C05422=1058.891,318.476,-103.732,173.436,35.812,156.715
C05423=1058.885,318.224,-103.698,173.433,35.808,156.714
C05424=1058.878,317.971,-103.663,173.428,35.803,156.713
C05425=1058.871,317.718,-103.629,173.425,35.799,156.712
C05426=1058.864,317.467,-103.595,173.421,35.795,156.711
C05427=1058.859,317.219,-103.561,173.418,35.790,156.711
C05428=1058.852,316.971,-103.527,173.414,35.786,156.710
C05429=1058.846,316.723,-103.494,173.411,35.782,156.709
C05430=1058.839,316.476,-103.460,173.408,35.778,156.708
C05431=1058.833,316.228,-103.426,173.404,35.773,156.707
C05432=1058.827,315.981,-103.393,173.401,35.769,156.706
C05433=1058.820,315.733,-103.359,173.397,35.765,156.705
C05434=1058.814,315.485,-103.326,173.394,35.760,156.704
C05435=1058.808,315.238,-103.292,173.391,35.756,156.703
C05436=1058.801,314.989,-103.259,173.388,35.752,156.702
C05437=1058.795,314.742,-103.225,173.384,35.748,156.701
C05438=1058.789,314.495,-103.192,173.381,35.744,156.700
C05439=1058.783,314.247,-103.158,173.378,35.740,156.699
C05440=1058.776,313.999,-103.125,173.374,35.735,156.698
C05441=1058.770,313.752,-103.091,173.371,35.731,156.698
C05442=1058.763,313.503,-103.058,173.367,35.727,156.697
C05443=1058.757,313.256,-103.025,173.364,35.723,156.696
C05444=1058.751,313.009,-102.992,173.360,35.719,156.695
C05445=1058.744,312.761,-102.959,173.357,35.715,156.694
C05446=1058.737,312.513,-102.926,173.354,35.711,156.693
C05447=1058.730,312.265,-102.892,173.350,35.706,156.692
C05448=1058.724,312.018,-102.859,173.347,35.702,156.691
C05449=1058.717,311.770,-102.827,173.343,35.698,156.691
C05450=1058.710,311.522,-102.794,173.340,35.694,156.690
C05451=1058.704,311.275,-102.761,173.337,35.690,156.689
C05452=1058.697,311.028,-102.728,173.333,35.686,156.688
C05453=1058.690,310.779,-102.695,173.330,35.682,156.687
C05454=1058.684,310.532,-102.662,173.326,35.678,156.686
C05455=1058.678,310.284,-102.629,173.323,35.674,156.685
C05456=1058.671,310.036,-102.596,173.320,35.670,156.684
C05457=1058.664,309.788,-102.563,173.316,35.666,156.684
C05458=1058.658,309.541,-102.531,173.314,35.662,156.683
C05459=1058.652,309.293,-102.498,173.310,35.658,156.682
C05460=1058.645,309.045,-102.465,173.307,35.654,156.681
C05461=1058.639,308.797,-102.432,173.303,35.650,156.680
C05462=1058.631,308.551,-102.399,173.300,35.645,156.679
C05463=1058.625,308.302,-102.367,173.297,35.642,156.679
C05464=1058.618,308.054,-102.334,173.293,35.638,156.678
C05465=1058.612,307.806,-102.301,173.290,35.634,156.677
C05466=1058.606,307.559,-102.269,173.287,35.630,156.676
C05467=1058.600,307.311,-102.236,173.283,35.626,156.675
C05468=1058.593,307.064,-102.203,173.280,35.622,156.674
C05469=1058.586,306.815,-102.170,173.277,35.617,156.673
C05470=1058.579,306.568,-102.138,173.274,35.613,156.672
C05471=1058.573,306.320,-102.105,173.271,35.609,156.672
C05472=1058.567,306.073,-102.072,173.267,35.605,156.671
C05473=1058.560,305.825,-102.040,173.264,35.601,156.670
C05474=1058.554,305.578,-102.007,173.260,35.598,156.669
C05475=1058.548,305.329,-101.975,173.257,35.594,156.668
C05476=1058.541,305.081,-101.942,173.255,35.590,156.667
C05477=1058.534,304.834,-101.910,173.251,35.585,156.666
C05478=1058.528,304.586,-101.877,173.248,35.581,156.666
C05479=1058.522,304.338,-101.845,173.244,35.577,156.665
C05480=1058.515,304.090,-101.812,173.241,35.573,156.664
C05481=1058.509,303.842,-101.780,173.238,35.569,156.663
C05482=1058.503,303.593,-101.746,173.234,35.566,156.662
C05483=1058.496,303.345,-101.715,173.232,35.561,156.661
C05484=1058.490,303.097,-101.682,173.228,35.557,156.660
C05485=1058.484,302.850,-101.649,173.225,35.553,156.660
C05486=1058.478,302.602,-101.617,173.222,35.549,156.659
C05487=1058.471,302.354,-101.584,173.218,35.545,156.658
C05488=1058.464,302.107,-101.552,173.216,35.541,156.657
C05489=1058.458,301.859,-101.520,173.213,35.538,156.656
C05490=1058.452,301.611,-101.487,173.209,35.533,156.655
C05491=1058.446,301.363,-101.455,173.206,35.529,156.655
C05492=1058.440,301.115,-101.423,173.202,35.525,156.654
C05493=1058.433,300.867,-101.391,173.200,35.521,156.653
C05494=1058.427,300.620,-101.358,173.197,35.517,156.652
C05495=1058.420,300.372,-101.326,173.193,35.514,156.651
C05496=1058.414,300.124,-101.294,173.190,35.509,156.650
C05497=1058.408,299.876,-101.261,173.187,35.505,156.649
C05498=1058.401,299.628,-101.230,173.184,35.501,156.649
C05499=1058.395,299.380,-101.198,173.181,35.497,156.648
C05500=1058.389,299.133,-101.165,173.177,35.494,156.647
C05501=1058.383,298.884,-101.133,173.174,35.490,156.646
C05502=1058.377,298.638,-101.101,173.172,35.485,156.645
C05503=1058.371,298.390,-101.069,173.168,35.481,156.644
C05504=1058.364,298.142,-101.036,173.165,35.477,156.644
C05505=1058.358,297.894,-101.004,173.162,35.474,156.643
C05506=1058.352,297.646,-100.973,173.159,35.470,156.642
C05507=1058.345,297.398,-100.940,173.156,35.466,156.641
C05508=1058.339,297.150,-100.908,173.152,35.461,156.640
C05509=1058.334,296.903,-100.876,173.150,35.457,156.639
C05510=1058.327,296.655,-100.844,173.147,35.454,156.639
C05511=1058.321,296.407,-100.812,173.143,35.450,156.638
C05512=1058.314,296.159,-100.781,173.140,35.446,156.637
C05513=1058.308,295.911,-100.749,173.138,35.442,156.636
C05514=1058.302,295.663,-100.717,173.134,35.438,156.635
C05515=1058.295,295.415,-100.685,173.131,35.434,156.635
C05516=1058.289,295.168,-100.653,173.128,35.430,156.634
C05517=1058.283,294.919,-100.621,173.125,35.426,156.633
C05518=1058.276,294.672,-100.590,173.122,35.423,156.632
C05519=1058.270,294.424,-100.559,173.119,35.419,156.631
C05520=1058.264,294.176,-100.527,173.115,35.415,156.630
C05521=1058.257,293.928,-100.495,173.113,35.411,156.630
C05522=1058.250,293.680,-100.464,173.110,35.407,156.629
C05523=1058.244,293.432,-100.432,173.106,35.403,156.628
C05524=1058.238,293.185,-100.401,173.104,35.399,156.627
C05525=1058.232,292.937,-100.369,173.101,35.396,156.626
C05526=1058.226,292.689,-100.337,173.097,35.392,156.626
C05527=1058.219,292.441,-100.306,173.095,35.388,156.625
C05528=1058.213,292.193,-100.274,173.092,35.384,156.624
C05529=1058.206,291.945,-100.242,173.088,35.380,156.623
C05530=1058.200,291.697,-100.211,173.086,35.376,156.622
C05531=1058.194,291.457,-100.180,173.083,35.373,156.622
C05532=1058.188,291.217,-100.150,173.079,35.369,156.621
C05533=1058.182,290.976,-100.119,173.077,35.365,156.620
C05534=1058.175,290.736,-100.089,173.074,35.362,156.619
C05535=1058.169,290.496,-100.058,173.071,35.358,156.619
C05536=1058.163,290.255,-100.028,173.068,35.354,156.618
C05537=1058.156,290.015,-99.998,173.065,35.350,156.617
C05538=1058.151,289.774,-99.967,173.062,35.347,156.616
C05539=1058.144,289.527,-99.936,173.059,35.343,156.615
C05540=1058.138,289.279,-99.905,173.057,35.339,156.615
C05541=1058.132,289.031,-99.872,173.053,35.335,156.614
C05542=1058.126,288.783,-99.842,173.050,35.332,156.613
C05543=1058.119,288.535,-99.811,173.048,35.327,156.612
C05544=1058.112,288.287,-99.779,173.044,35.324,156.611
C05545=1058.106,288.039,-99.749,173.041,35.320,156.611
C05546=1058.100,287.791,-99.717,173.039,35.316,156.610
C05547=1058.094,287.543,-99.685,173.035,35.313,156.609
C05548=1058.088,287.295,-99.655,173.032,35.309,156.608
C05549=1058.081,287.047,-99.623,173.030,35.305,156.607
C05550=1058.075,286.800,-99.592,173.026,35.301,156.607
C05551=1058.068,286.551,-99.562,173.024,35.297,156.606
C05552=1058.062,286.303,-99.530,173.021,35.294,156.605
C05553=1058.056,286.055,-99.500,173.017,35.290,156.604
C05554=1058.049,285.807,-99.468,173.015,35.286,156.604
C05555=1058.042,285.560,-99.437,173.012,35.282,156.603
C05556=1058.036,285.312,-99.407,173.008,35.278,156.602
C05557=1058.030,285.064,-99.375,173.006,35.275,156.601
C05558=1058.023,284.815,-99.344,173.003,35.271,156.600
C05559=1058.017,284.568,-99.313,173.001,35.267,156.600
C05560=1058.011,284.320,-99.283,172.997,35.263,156.599
C05561=1058.004,284.071,-99.252,172.994,35.260,156.598
C05562=1057.998,283.824,-99.221,172.992,35.256,156.597
C05563=1057.992,283.575,-99.190,172.988,35.252,156.596
C05564=1057.986,283.328,-99.159,172.986,35.248,156.596
C05565=1057.979,283.080,-99.128,172.983,35.245,156.595
C05566=1057.973,282.832,-99.097,172.980,35.241,156.594
C05567=1057.967,282.584,-99.067,172.977,35.237,156.593
C05568=1057.960,282.335,-99.036,172.974,35.233,156.593
C05569=1057.954,282.088,-99.005,172.971,35.229,156.592
C05570=1057.948,281.840,-98.974,172.968,35.226,156.591
C05571=1057.942,281.592,-98.944,172.966,35.222,156.590
C05572=1057.935,281.344,-98.912,172.962,35.218,156.590
C05573=1057.929,281.096,-98.882,172.960,35.215,156.589
C05574=1057.923,280.848,-98.851,172.957,35.210,156.588
C05575=1057.917,280.600,-98.821,172.955,35.207,156.587
C05576=1057.910,280.352,-98.789,172.951,35.203,156.586
C05577=1057.905,280.104,-98.759,172.949,35.199,156.586
C05578=1057.898,279.856,-98.728,172.946,35.196,156.585
C05579=1057.892,279.608,-98.698,172.942,35.192,156.584
C05580=1057.885,279.359,-98.668,172.940,35.188,156.583
C05581=1057.879,279.112,-98.636,172.937,35.184,156.583
C05582=1057.873,278.864,-98.606,172.934,35.181,156.582
C05583=1057.866,278.615,-98.575,172.931,35.177,156.581
C05584=1057.860,278.368,-98.546,172.929,35.173,156.580
C05585=1057.853,278.119,-98.515,172.926,35.170,156.580
C05586=1057.847,277.871,-98.485,172.923,35.165,156.579
C05587=1057.842,277.637,-98.456,172.920,35.162,156.578
C05588=1057.836,277.401,-98.427,172.918,35.159,156.577
C05589=1057.830,277.166,-98.398,172.915,35.155,156.577
C05590=1057.824,276.932,-98.369,172.912,35.152,156.576
C05591=1057.817,276.697,-98.341,172.910,35.148,156.575
C05592=1057.811,276.462,-98.312,172.907,35.145,156.574
C05593=1057.806,276.227,-98.283,172.904,35.141,156.574
C05594=1057.800,275.992,-98.255,172.902,35.138,156.573
C05595=1057.794,275.744,-98.224,172.899,35.134,156.572
C05596=1057.787,275.496,-98.194,172.896,35.130,156.571
C05597=1057.781,275.248,-98.163,172.893,35.126,156.571
C05598=1057.775,275.000,-98.133,172.891,35.123,156.570
C05599=1057.764,274.601,-98.084,172.886,35.117,156.569
C05600=1057.754,274.203,-98.036,172.882,35.111,156.568
C05601=1057.744,273.805,-97.988,172.877,35.105,156.566
C05602=1057.734,273.406,-97.940,172.873,35.099,156.565
C05603=1057.728,273.158,-97.909,172.870,35.095,156.564
C05604=1057.722,272.911,-97.879,172.867,35.091,156.564
C05605=1057.715,272.662,-97.849,172.865,35.088,156.563
C05606=1057.710,272.414,-97.819,172.862,35.084,156.562
C05607=1057.703,272.166,-97.789,172.860,35.081,156.561
C05608=1057.697,271.918,-97.759,172.856,35.076,156.560
C05609=1057.690,271.670,-97.730,172.854,35.073,156.560
C05610=1057.684,271.421,-97.699,172.851,35.069,156.559
C05611=1057.678,271.173,-97.669,172.849,35.066,156.558
C05612=1057.672,270.926,-97.639,172.845,35.062,156.558
C05613=1057.665,270.677,-97.609,172.843,35.058,156.557
C05614=1057.659,270.429,-97.579,172.841,35.054,156.556
C05615=1057.653,270.181,-97.550,172.837,35.051,156.555
C05616=1057.646,269.933,-97.519,172.835,35.047,156.555
C05617=1057.640,269.685,-97.490,172.832,35.044,156.554
C05618=1057.634,269.437,-97.460,172.830,35.040,156.553
C05619=1057.627,269.188,-97.430,172.826,35.036,156.552
C05620=1057.621,268.940,-97.400,172.824,35.032,156.552
C05621=1057.615,268.692,-97.370,172.822,35.029,156.551
C05622=1057.609,268.444,-97.341,172.818,35.025,156.550
C05623=1057.602,268.196,-97.311,172.816,35.021,156.549
C05624=1057.596,267.948,-97.282,172.813,35.018,156.549
C05625=1057.590,267.700,-97.251,172.811,35.014,156.548
C05626=1057.583,267.451,-97.222,172.808,35.010,156.547
C05627=1057.577,267.204,-97.192,172.805,35.007,156.546
C05628=1057.571,266.955,-97.162,172.803,35.003,156.546
C05629=1057.565,266.708,-97.133,172.800,35.000,156.545
C05630=1057.558,266.459,-97.103,172.797,34.995,156.544
C05631=1057.552,266.210,-97.074,172.795,34.992,156.543
C05632=1057.546,265.963,-97.044,172.792,34.988,156.543
C05633=1057.540,265.715,-97.015,172.790,34.985,156.542
C05634=1057.533,265.466,-96.984,172.786,34.981,156.541
C05635=1057.527,265.218,-96.955,172.784,34.978,156.540
C05636=1057.521,264.970,-96.926,172.782,34.973,156.540
C05637=1057.515,264.722,-96.896,172.778,34.970,156.539
C05638=1057.509,264.474,-96.867,172.776,34.966,156.538
C05639=1057.502,264.225,-96.837,172.774,34.963,156.537
C05640=1057.496,263.977,-96.808,172.771,34.959,156.537
C05641=1057.490,263.729,-96.778,172.768,34.956,156.536
C05642=1057.483,263.481,-96.749,172.766,34.951,156.535
C05643=1057.476,263.165,-96.712,172.763,34.947,156.534
C05644=1057.468,262.850,-96.674,172.760,34.942,156.533
C05645=1057.460,262.534,-96.637,172.756,34.938,156.532
C05646=1057.451,262.219,-96.600,172.753,34.933,156.532
C05647=1057.444,261.971,-96.570,172.750,34.930,156.531
C05648=1057.438,261.722,-96.541,172.747,34.926,156.530
C05649=1057.432,261.474,-96.512,172.745,34.923,156.529
C05650=1057.425,261.226,-96.483,172.742,34.919,156.529
C05651=1057.418,260.977,-96.454,172.740,34.915,156.528
C05652=1057.412,260.729,-96.425,172.737,34.912,156.527
C05653=1057.406,260.481,-96.396,172.734,34.908,156.526
C05654=1057.400,260.233,-96.367,172.732,34.905,156.526
C05655=1057.393,259.985,-96.338,172.730,34.901,156.525
C05656=1057.387,259.737,-96.309,172.726,34.897,156.524
C05657=1057.380,259.488,-96.279,172.724,34.893,156.523
C05658=1057.374,259.240,-96.250,172.722,34.890,156.523
C05659=1057.368,258.992,-96.221,172.719,34.886,156.522
C05660=1057.362,258.743,-96.192,172.716,34.883,156.521
C05661=1057.355,258.495,-96.163,172.714,34.879,156.521
C05662=1057.349,258.247,-96.134,172.711,34.875,156.520
C05663=1057.343,257.999,-96.105,172.709,34.872,156.519
C05664=1057.336,257.751,-96.077,172.706,34.868,156.518
C05665=1057.329,257.502,-96.047,172.703,34.865,156.518
C05666=1057.323,257.254,-96.019,172.701,34.861,156.517
C05667=1057.317,257.006,-95.990,172.699,34.857,156.516
C05668=1057.311,256.757,-95.961,172.695,34.854,156.516
C05669=1057.304,256.509,-95.932,172.693,34.850,156.515
C05670=1057.298,256.261,-95.903,172.691,34.847,156.514
C05671=1057.292,256.013,-95.874,172.689,34.843,156.513
C05672=1057.286,255.765,-95.845,172.685,34.839,156.513
C05673=1057.280,255.516,-95.816,172.683,34.836,156.512
C05674=1057.273,255.268,-95.787,172.681,34.832,156.511
C05675=1057.266,255.020,-95.759,172.679,34.828,156.510
C05676=1057.260,254.772,-95.730,172.675,34.825,156.510
C05677=1057.254,254.523,-95.701,172.673,34.821,156.509
C05678=1057.248,254.275,-95.672,172.671,34.817,156.508
C05679=1057.242,254.027,-95.643,172.669,34.814,156.508
C05680=1057.235,253.779,-95.614,172.666,34.810,156.507
C05681=1057.230,253.530,-95.586,172.663,34.807,156.506
C05682=1057.223,253.282,-95.557,172.661,34.803,156.505
C05683=1057.217,253.034,-95.528,172.659,34.799,156.505
C05684=1057.210,252.785,-95.500,172.656,34.796,156.504
C05685=1057.204,252.537,-95.471,172.653,34.792,156.503
C05686=1057.198,252.289,-95.443,172.651,34.788,156.502
C05687=1057.192,252.040,-95.414,172.649,34.784,156.502
C05688=1057.186,251.792,-95.385,172.646,34.781,156.501
C05689=1057.180,251.544,-95.356,172.643,34.777,156.500
C05690=1057.173,251.295,-95.327,172.641,34.774,156.500
C05691=1057.167,251.047,-95.300,172.639,34.770,156.499
C05692=1057.161,250.799,-95.271,172.637,34.766,156.498
C05693=1057.155,250.551,-95.242,172.633,34.762,156.497
C05694=1057.149,250.303,-95.214,172.631,34.759,156.497
C05695=1057.143,250.068,-95.186,172.629,34.755,156.496
C05696=1057.137,249.835,-95.159,172.627,34.752,156.495
C05697=1057.131,249.601,-95.132,172.625,34.748,156.494
C05698=1057.125,249.367,-95.106,172.622,34.745,156.494
C05699=1057.120,249.133,-95.079,172.620,34.741,156.493
C05700=1057.114,248.900,-95.052,172.618,34.738,156.492
C05701=1057.108,248.665,-95.025,172.616,34.735,156.492
C05702=1057.103,248.431,-94.998,172.613,34.731,156.491
C05703=1057.096,248.183,-94.970,172.611,34.727,156.490
C05704=1057.090,247.935,-94.942,172.608,34.724,156.490
C05705=1057.084,247.686,-94.913,172.606,34.720,156.489
C05706=1057.078,247.438,-94.884,172.604,34.716,156.488
C05707=1057.072,247.189,-94.856,172.601,34.712,156.487
C05708=1057.066,246.941,-94.828,172.599,34.709,156.487
C05709=1057.060,246.694,-94.799,172.597,34.705,156.486
C05710=1057.054,246.445,-94.771,172.594,34.701,156.485
C05711=1057.048,246.196,-94.743,172.591,34.697,156.484
C05712=1057.041,245.948,-94.714,172.589,34.694,156.484
C05713=1057.035,245.699,-94.686,172.587,34.690,156.483
C05714=1057.029,245.451,-94.658,172.585,34.687,156.482
C05715=1057.023,245.203,-94.630,172.583,34.683,156.481
C05716=1057.017,244.955,-94.601,172.579,34.679,156.481
C05717=1057.010,244.706,-94.574,172.577,34.676,156.480
C05718=1057.004,244.458,-94.545,172.575,34.672,156.479
C05719=1056.998,244.209,-94.517,172.573,34.668,156.479
C05720=1056.992,243.961,-94.490,172.570,34.664,156.478
C05721=1056.986,243.713,-94.461,172.568,34.661,156.477
C05722=1056.979,243.465,-94.433,172.566,34.657,156.476
C05723=1056.973,243.216,-94.404,172.563,34.654,156.476
C05724=1056.967,242.967,-94.377,172.561,34.650,156.475
C05725=1056.961,242.719,-94.349,172.558,34.646,156.474
C05726=1056.955,242.471,-94.321,172.556,34.643,156.474
C05727=1056.949,242.222,-94.293,172.554,34.639,156.473
C05728=1056.942,241.974,-94.264,172.552,34.635,156.472
C05729=1056.936,241.726,-94.236,172.549,34.631,156.471
C05730=1056.930,241.478,-94.209,172.547,34.628,156.471
C05731=1056.924,241.229,-94.180,172.544,34.624,156.470
C05732=1056.917,240.981,-94.153,172.542,34.620,156.469
C05733=1056.911,240.733,-94.125,172.540,34.617,156.468
C05734=1056.905,240.484,-94.097,172.537,34.613,156.468
C05735=1056.898,240.236,-94.069,172.535,34.610,156.467
C05736=1056.892,239.987,-94.041,172.533,34.606,156.466
C05737=1056.886,239.739,-94.013,172.531,34.602,156.466
C05738=1056.880,239.490,-93.986,172.529,34.599,156.465
C05739=1056.873,239.242,-93.959,172.526,34.595,156.464
C05740=1056.867,238.993,-93.930,172.523,34.592,156.463
C05741=1056.861,238.745,-93.903,172.521,34.588,156.463
C05742=1056.854,238.497,-93.875,172.519,34.584,156.462
C05743=1056.849,238.248,-93.847,172.516,34.580,156.461
C05744=1056.842,238.000,-93.819,172.514,34.577,156.460
C05745=1056.836,237.752,-93.792,172.512,34.573,156.460
C05746=1056.829,237.503,-93.764,172.510,34.569,156.459
C05747=1056.823,237.254,-93.736,172.508,34.566,156.458
C05748=1056.817,237.006,-93.709,172.505,34.562,156.458
C05749=1056.811,236.758,-93.681,172.503,34.558,156.457
C05750=1056.804,236.509,-93.654,172.501,34.555,156.456
C05751=1056.799,236.273,-93.628,172.499,34.551,156.455
C05752=1056.792,236.036,-93.601,172.497,34.548,156.455
C05753=1056.787,235.799,-93.574,172.494,34.544,156.454
C05754=1056.781,235.562,-93.548,172.492,34.541,156.453
C05755=1056.775,235.325,-93.522,172.490,34.537,156.453
C05756=1056.769,235.088,-93.495,172.488,34.534,156.452
C05757=1056.763,234.850,-93.470,172.486,34.530,156.451
C05758=1056.758,234.614,-93.444,172.484,34.527,156.451
C05759=1056.751,234.365,-93.416,172.481,34.523,156.450
C05760=1056.744,234.117,-93.388,172.479,34.519,156.449
C05761=1056.739,233.868,-93.361,172.477,34.516,156.448
C05762=1056.732,233.620,-93.333,172.475,34.512,156.448
C05763=1056.726,233.372,-93.306,172.473,34.508,156.447
C05764=1056.720,233.123,-93.279,172.470,34.504,156.446
C05765=1056.714,232.875,-93.252,172.468,34.501,156.446
C05766=1056.708,232.627,-93.223,172.466,34.497,156.445
C05767=1056.702,232.377,-93.196,172.464,34.493,156.444
C05768=1056.696,232.130,-93.169,172.462,34.490,156.443
C05769=1056.689,231.881,-93.142,172.459,34.486,156.443
C05770=1056.683,231.633,-93.115,172.457,34.483,156.442
C05771=1056.677,231.384,-93.088,172.455,34.479,156.441
C05772=1056.670,231.135,-93.060,172.453,34.475,156.440
C05773=1056.664,230.887,-93.033,172.451,34.471,156.440
C05774=1056.658,230.639,-93.005,172.448,34.467,156.439
C05775=1056.652,230.390,-92.979,172.446,34.464,156.438
C05776=1056.645,230.142,-92.951,172.444,34.460,156.438
C05777=1056.639,229.893,-92.924,172.442,34.457,156.437
C05778=1056.633,229.645,-92.896,172.440,34.453,156.436
C05779=1056.628,229.396,-92.869,172.437,34.449,156.435
C05780=1056.621,229.148,-92.842,172.435,34.445,156.435
C05781=1056.614,228.900,-92.816,172.433,34.441,156.434
C05782=1056.608,228.651,-92.788,172.431,34.438,156.433
C05783=1056.601,228.402,-92.761,172.429,34.434,156.433
C05784=1056.596,228.154,-92.734,172.426,34.431,156.432
C05785=1056.589,227.906,-92.706,172.424,34.427,156.431
C05786=1056.583,227.657,-92.680,172.422,34.423,156.430
C05787=1056.577,227.408,-92.653,172.420,34.420,156.430
C05788=1056.570,227.161,-92.626,172.418,34.416,156.429
C05789=1056.564,226.912,-92.599,172.415,34.412,156.428
C05790=1056.558,226.663,-92.572,172.413,34.408,156.427
C05791=1056.551,226.415,-92.545,172.411,34.405,156.427
C05792=1056.545,226.167,-92.518,172.409,34.401,156.426
C05793=1056.539,225.917,-92.491,172.407,34.397,156.425
C05794=1056.533,225.669,-92.464,172.405,34.394,156.425
C05795=1056.526,225.421,-92.437,172.402,34.390,156.424
C05796=1056.520,225.173,-92.411,172.400,34.386,156.423
C05797=1056.514,224.924,-92.384,172.398,34.383,156.422
C05798=1056.508,224.675,-92.357,172.396,34.379,156.422
C05799=1056.502,224.427,-92.330,172.394,34.375,156.421
C05800=1056.495,224.178,-92.303,172.391,34.371,156.420
C05801=1056.489,223.930,-92.276,172.389,34.368,156.420
C05802=1056.482,223.681,-92.249,172.387,34.364,156.419
C05803=1056.477,223.433,-92.223,172.385,34.360,156.418
C05804=1056.471,223.185,-92.196,172.383,34.356,156.417
C05805=1056.465,222.935,-92.169,172.382,34.353,156.417
C05806=1056.459,222.687,-92.143,172.379,34.349,156.416
C05807=1056.452,222.446,-92.116,172.377,34.345,156.415
C05808=1056.447,222.206,-92.090,172.375,34.342,156.414
C05809=1056.440,221.964,-92.064,172.373,34.338,156.414
C05810=1056.434,221.724,-92.038,172.371,34.335,156.413
C05811=1056.428,221.483,-92.012,172.368,34.331,156.412
C05812=1056.423,221.242,-91.987,172.366,34.327,156.412
C05813=1056.416,221.001,-91.961,172.365,34.324,156.411
C05814=1056.411,220.760,-91.935,172.363,34.320,156.410
C05815=1056.404,220.512,-91.909,172.361,34.316,156.410
C05816=1056.398,220.263,-91.882,172.359,34.313,156.409
C05817=1056.391,220.015,-91.856,172.356,34.309,156.408
C05818=1056.385,219.766,-91.829,172.354,34.305,156.407
C05819=1056.379,219.518,-91.803,172.352,34.301,156.407
C05820=1056.372,219.269,-91.776,172.350,34.298,156.406
C05821=1056.366,219.021,-91.750,172.348,34.294,156.405
C05822=1056.360,218.773,-91.724,172.347,34.290,156.404
C05823=1056.353,218.524,-91.696,172.344,34.287,156.404
C05824=1056.347,218.276,-91.670,172.342,34.283,156.403
C05825=1056.341,218.027,-91.644,172.340,34.279,156.402
C05826=1056.335,217.778,-91.617,172.338,34.275,156.402
C05827=1056.329,217.530,-91.591,172.336,34.272,156.401
C05828=1056.323,217.281,-91.565,172.334,34.268,156.400
C05829=1056.316,217.032,-91.538,172.331,34.264,156.399
C05830=1056.310,216.784,-91.512,172.329,34.260,156.399
C05831=1056.303,216.536,-91.486,172.328,34.257,156.398
C05832=1056.297,216.287,-91.459,172.326,34.253,156.397
C05833=1056.291,216.038,-91.433,172.324,34.249,156.396
C05834=1056.285,215.790,-91.407,172.321,34.246,156.396
C05835=1056.279,215.542,-91.381,172.319,34.241,156.395
C05836=1056.272,215.293,-91.354,172.317,34.238,156.394
C05837=1056.266,215.044,-91.328,172.315,34.234,156.394
C05838=1056.260,214.796,-91.302,172.314,34.230,156.393
C05839=1056.254,214.548,-91.276,172.312,34.226,156.392
C05840=1056.247,214.299,-91.249,172.309,34.223,156.391
C05841=1056.241,214.050,-91.223,172.307,34.219,156.391
C05842=1056.235,213.802,-91.197,172.305,34.215,156.390
C05843=1056.229,213.554,-91.171,172.303,34.211,156.389
C05844=1056.223,213.304,-91.144,172.302,34.207,156.388
C05845=1056.217,213.056,-91.118,172.300,34.204,156.388
C05846=1056.210,212.808,-91.092,172.297,34.200,156.387
C05847=1056.204,212.559,-91.066,172.295,34.196,156.386
C05848=1056.198,212.311,-91.040,172.293,34.192,156.385
C05849=1056.191,212.062,-91.013,172.291,34.189,156.385
C05850=1056.186,211.813,-90.987,172.290,34.184,156.384
C05851=1056.179,211.565,-90.961,172.288,34.181,156.383
C05852=1056.173,211.316,-90.936,172.286,34.177,156.383
C05853=1056.167,211.067,-90.909,172.283,34.174,156.382
C05854=1056.160,210.819,-90.883,172.281,34.169,156.381
C05855=1056.154,210.570,-90.857,172.279,34.166,156.380
C05856=1056.148,210.322,-90.831,172.278,34.162,156.380
C05857=1056.142,210.073,-90.805,172.276,34.158,156.379
C05858=1056.135,209.824,-90.779,172.274,34.154,156.378
C05859=1056.129,209.576,-90.753,172.271,34.150,156.377
C05860=1056.123,209.327,-90.727,172.269,34.147,156.377
C05861=1056.117,209.079,-90.702,172.268,34.143,156.376
C05862=1056.110,208.831,-90.676,172.266,34.139,156.375
C05863=1056.104,208.592,-90.650,172.264,34.135,156.374
C05864=1056.099,208.354,-90.625,172.262,34.132,156.374
C05865=1056.092,208.116,-90.601,172.260,34.128,156.373
C05866=1056.087,207.877,-90.576,172.258,34.124,156.372
C05867=1056.081,207.639,-90.552,172.256,34.121,156.372
C05868=1056.075,207.400,-90.527,172.255,34.117,156.371
C05869=1056.069,207.162,-90.502,172.253,34.114,156.370
C05870=1056.062,206.924,-90.478,172.251,34.110,156.370
C05871=1056.037,205.873,-90.373,172.050,34.020,156.356
C05872=1056.031,205.624,-90.348,172.048,34.017,156.356
C05873=1056.025,205.376,-90.323,172.045,34.014,156.355
C05874=1056.020,205.127,-90.298,172.043,34.011,156.355
C05875=1056.013,204.878,-90.273,172.041,34.008,156.354
C05876=1056.008,204.630,-90.248,172.038,34.005,156.354
C05877=1056.001,204.381,-90.224,172.036,34.002,156.353
C05878=1055.996,204.133,-90.199,172.034,33.999,156.353
C05879=1055.990,203.884,-90.174,172.031,33.996,156.352
C05880=1055.984,203.635,-90.149,172.028,33.993,156.352
C05881=1055.978,203.387,-90.124,172.026,33.990,156.351
C05882=1055.972,203.138,-90.100,172.024,33.987,156.351
C05883=1055.966,202.888,-90.075,172.021,33.984,156.350
C05884=1055.961,202.640,-90.050,172.019,33.982,156.350
C05885=1055.954,202.391,-90.026,172.017,33.978,156.349
C05886=1055.948,202.143,-90.001,172.015,33.975,156.348
C05887=1055.943,201.894,-89.977,172.012,33.972,156.348
C05888=1055.937,201.645,-89.952,172.010,33.970,156.347
C05889=1055.930,201.397,-89.928,172.008,33.967,156.347
C05890=1055.924,201.148,-89.903,172.005,33.964,156.346
C05891=1055.918,200.899,-89.878,172.002,33.961,156.346
C05892=1055.912,200.651,-89.854,172.000,33.958,156.345
C05893=1055.906,200.402,-89.829,171.998,33.955,156.345
C05894=1055.900,200.153,-89.806,171.995,33.953,156.344
C05895=1055.894,199.904,-89.781,171.993,33.950,156.344
C05896=1055.888,199.655,-89.756,171.991,33.947,156.343
C05897=1055.882,199.407,-89.732,171.989,33.944,156.343
C05898=1055.876,199.158,-89.707,171.986,33.941,156.342
C05899=1055.870,198.910,-89.684,171.984,33.938,156.342
C05900=1055.864,198.661,-89.658,171.982,33.936,156.341
C05901=1055.857,198.412,-89.634,171.980,33.933,156.341
C05902=1055.852,198.163,-89.610,171.976,33.930,156.340
C05903=1055.845,197.914,-89.586,171.974,33.927,156.340
C05904=1055.840,197.666,-89.562,171.972,33.924,156.339
C05905=1055.834,197.416,-89.537,171.970,33.921,156.339
C05906=1055.828,197.169,-89.513,171.967,33.919,156.338
C05907=1055.822,196.919,-89.488,171.965,33.916,156.338
C05908=1055.815,196.671,-89.464,171.963,33.913,156.337
C05909=1055.810,196.422,-89.440,171.961,33.910,156.337
C05910=1055.803,196.173,-89.416,171.958,33.907,156.336
C05911=1055.798,195.924,-89.392,171.956,33.904,156.336
C05912=1055.791,195.675,-89.368,171.954,33.902,156.335
C05913=1055.786,195.427,-89.343,171.952,33.899,156.335
C05914=1055.779,195.178,-89.319,171.949,33.896,156.334
C05915=1055.774,194.929,-89.295,171.946,33.893,156.334
C05916=1055.768,194.680,-89.271,171.944,33.891,156.333
C05917=1055.762,194.432,-89.247,171.942,33.887,156.333
C05918=1055.756,194.183,-89.223,171.940,33.885,156.332
C05919=1055.750,193.934,-89.199,171.937,33.882,156.332
C05920=1055.744,193.686,-89.175,171.935,33.879,156.331
C05921=1055.738,193.437,-89.150,171.933,33.876,156.331
C05922=1055.732,193.188,-89.127,171.931,33.874,156.330
C05923=1055.726,192.939,-89.102,171.929,33.870,156.330
C05924=1055.720,192.691,-89.078,171.926,33.868,156.329
C05925=1055.714,192.441,-89.054,171.924,33.865,156.329
C05926=1055.708,192.193,-89.030,171.922,33.862,156.328
C05927=1055.703,191.945,-89.006,171.920,33.860,156.328
C05928=1055.696,191.696,-88.982,171.917,33.857,156.327
C05929=1055.691,191.447,-88.958,171.915,33.854,156.327
C05930=1055.685,191.198,-88.933,171.912,33.851,156.326
C05931=1055.679,190.949,-88.909,171.910,33.848,156.326
C05932=1055.673,190.665,-88.882,171.908,33.845,156.325
C05933=1055.666,190.381,-88.855,171.905,33.842,156.325
C05934=1055.659,190.097,-88.827,171.903,33.839,156.324
C05935=1055.653,189.813,-88.800,171.900,33.836,156.323
C05936=1055.647,189.564,-88.777,171.898,33.833,156.323
C05937=1055.641,189.316,-88.752,171.896,33.830,156.322
C05938=1055.635,189.067,-88.728,171.894,33.827,156.322
C05939=1055.630,188.818,-88.705,171.892,33.824,156.321
C05940=1055.624,188.569,-88.681,171.890,33.822,156.321
C05941=1055.618,188.320,-88.656,171.887,33.819,156.320
C05942=1055.612,188.072,-88.633,171.884,33.816,156.320
C05943=1055.606,187.824,-88.609,171.882,33.813,156.319
C05944=1055.600,187.574,-88.585,171.880,33.811,156.319
C05945=1055.594,187.325,-88.562,171.878,33.807,156.318
C05946=1055.589,187.077,-88.537,171.876,33.805,156.318
C05947=1055.583,186.828,-88.514,171.874,33.802,156.317
C05948=1055.577,186.579,-88.490,171.871,33.799,156.317
C05949=1055.571,186.330,-88.466,171.869,33.797,156.316
C05950=1055.566,186.081,-88.442,171.867,33.794,156.316
C05951=1055.559,185.832,-88.418,171.865,33.791,156.315
C05952=1055.553,185.584,-88.395,171.863,33.788,156.315
C05953=1055.548,185.335,-88.371,171.861,33.785,156.314
C05954=1055.542,185.086,-88.348,171.859,33.783,156.314
C05955=1055.537,184.838,-88.323,171.857,33.780,156.313
C05956=1055.531,184.588,-88.300,171.854,33.777,156.313
C05957=1055.525,184.340,-88.276,171.851,33.774,156.312
C05958=1055.520,184.091,-88.253,171.849,33.771,156.312
C05959=1055.513,183.842,-88.229,171.847,33.769,156.311
C05960=1055.507,183.593,-88.206,171.845,33.766,156.311
C05961=1055.500,183.345,-88.183,171.843,33.764,156.311
C05962=1055.494,183.095,-88.159,171.841,33.761,156.310
C05963=1055.488,182.847,-88.136,171.839,33.759,156.310
C05964=1055.482,182.598,-88.113,171.837,33.756,156.309
C05965=1055.476,182.349,-88.089,171.834,33.754,156.309
C05966=1055.470,182.100,-88.066,171.832,33.751,156.308
C05967=1055.464,181.851,-88.043,171.830,33.748,156.308
C05968=1055.458,181.602,-88.019,171.828,33.745,156.307
C05969=1055.452,181.353,-87.996,171.826,33.743,156.307
C05970=1055.446,181.105,-87.972,171.824,33.740,156.306
C05971=1055.440,180.856,-87.949,171.822,33.738,156.306
C05972=1055.434,180.607,-87.926,171.820,33.735,156.306
C05973=1055.428,180.358,-87.902,171.817,33.733,156.305
C05974=1055.421,180.110,-87.880,171.814,33.730,156.305
C05975=1055.415,179.860,-87.857,171.812,33.727,156.304
C05976=1055.409,179.612,-87.833,171.810,33.725,156.304
C05977=1055.403,179.363,-87.810,171.808,33.722,156.303
C05978=1055.397,179.114,-87.787,171.806,33.719,156.303
C05979=1055.391,178.865,-87.763,171.804,33.717,156.302
C05980=1055.385,178.616,-87.740,171.802,33.714,156.302
C05981=1055.379,178.367,-87.717,171.800,33.712,156.301
C05982=1055.374,178.119,-87.694,171.798,33.709,156.301
C05983=1055.366,177.870,-87.671,171.796,33.707,156.301
C05984=1055.361,177.621,-87.648,171.793,33.704,156.300
C05985=1055.355,177.372,-87.625,171.791,33.702,156.300
C05986=1055.349,177.123,-87.602,171.789,33.698,156.299
C05987=1055.343,176.875,-87.578,171.787,33.696,156.299
C05988=1055.337,176.625,-87.555,171.785,33.693,156.298
C05989=1055.331,176.376,-87.532,171.783,33.691,156.298
C05990=1055.325,176.127,-87.509,171.781,33.688,156.297
C05991=1055.319,175.879,-87.487,171.779,33.686,156.297
C05992=1055.313,175.631,-87.463,171.777,33.683,156.296
C05993=1055.307,175.382,-87.440,171.774,33.681,156.296
C05994=1055.301,175.132,-87.417,171.772,33.678,156.296
C05995=1055.295,174.883,-87.394,171.770,33.676,156.295
C05996=1055.288,174.599,-87.368,171.767,33.672,156.295
C05997=1055.282,174.315,-87.341,171.765,33.669,156.294
C05998=1055.275,174.030,-87.316,171.763,33.667,156.294
C05999=1055.268,173.746,-87.289,171.760,33.664,156.293
C06000=1055.262,173.497,-87.266,171.758,33.661,156.293
C06001=1055.256,173.249,-87.243,171.756,33.658,156.292
C06002=1055.250,173.000,-87.220,171.754,33.656,156.292
C06003=1055.244,172.750,-87.197,171.752,33.653,156.291
C06004=1055.238,172.501,-87.174,171.750,33.651,156.291
C06005=1055.232,172.253,-87.152,171.748,33.648,156.290
C06006=1055.226,172.004,-87.129,171.746,33.645,156.290
C06007=1055.220,171.755,-87.106,171.744,33.643,156.289
C06008=1055.215,171.506,-87.083,171.742,33.640,156.289
C06009=1055.209,171.257,-87.060,171.740,33.638,156.288
C06010=1055.202,171.008,-87.038,171.738,33.635,156.288
C06011=1055.197,170.760,-87.015,171.736,33.632,156.288
C06012=1055.191,170.511,-86.992,171.734,33.630,156.287
C06013=1055.185,170.262,-86.969,171.732,33.627,156.287
C06014=1055.179,170.013,-86.946,171.729,33.625,156.286
C06015=1055.174,169.764,-86.923,171.727,33.622,156.286
C06016=1055.167,169.515,-86.901,171.725,33.620,156.285
C06017=1055.162,169.266,-86.878,171.723,33.617,156.285
C06018=1055.156,169.018,-86.855,171.721,33.615,156.284
C06019=1055.150,168.769,-86.832,171.719,33.611,156.284
C06020=1055.145,168.519,-86.809,171.717,33.609,156.283
C06021=1055.138,168.271,-86.787,171.715,33.606,156.283
C06022=1055.132,168.022,-86.764,171.713,33.604,156.283
C06023=1055.127,167.773,-86.741,171.711,33.601,156.282
C06024=1055.121,167.524,-86.718,171.709,33.599,156.282
C06025=1055.115,167.275,-86.696,171.707,33.596,156.281
C06026=1055.109,167.026,-86.673,171.705,33.594,156.281
C06027=1055.103,166.777,-86.651,171.703,33.591,156.280
C06028=1055.098,166.528,-86.628,171.701,33.589,156.280
C06029=1055.092,166.279,-86.605,171.699,33.586,156.280
C06030=1055.085,166.030,-86.583,171.697,33.583,156.279
C06031=1055.080,165.782,-86.560,171.695,33.581,156.279
C06032=1055.074,165.532,-86.537,171.693,33.578,156.278
C06033=1055.069,165.283,-86.514,171.692,33.575,156.278
C06034=1055.063,165.035,-86.492,171.690,33.573,156.277
C06035=1055.057,164.786,-86.469,171.688,33.570,156.277
C06036=1055.052,164.537,-86.447,171.686,33.568,156.276
C06037=1055.046,164.288,-86.424,171.683,33.565,156.276
C06038=1055.039,164.039,-86.402,171.681,33.563,156.275
C06039=1055.034,163.790,-86.379,171.679,33.560,156.275
C06040=1055.028,163.541,-86.357,171.677,33.557,156.275
C06041=1055.022,163.292,-86.334,171.675,33.555,156.274
C06042=1055.016,163.043,-86.311,171.673,33.552,156.274
C06043=1055.011,162.795,-86.290,171.671,33.550,156.273
C06044=1055.005,162.546,-86.267,171.669,33.547,156.273
C06045=1054.999,162.297,-86.244,171.667,33.545,156.272
C06046=1054.994,162.048,-86.222,171.665,33.542,156.272
C06047=1054.988,161.799,-86.199,171.663,33.539,156.271
C06048=1054.982,161.550,-86.176,171.661,33.536,156.271
C06049=1054.976,161.301,-86.155,171.659,33.534,156.270
C06050=1054.971,161.052,-86.132,171.658,33.531,156.270
C06051=1054.965,160.803,-86.110,171.656,33.529,156.270
C06052=1054.959,160.554,-86.087,171.654,33.526,156.269
C06053=1054.953,160.305,-86.065,171.652,33.524,156.269
C06054=1054.947,160.056,-86.043,171.650,33.521,156.268
C06055=1054.941,159.807,-86.021,171.648,33.519,156.268
C06056=1054.935,159.558,-85.998,171.646,33.517,156.267
C06057=1054.929,159.309,-85.977,171.644,33.514,156.267
C06058=1054.922,159.060,-85.954,171.642,33.512,156.267
C06059=1054.918,158.812,-85.932,171.640,33.509,156.266
C06060=1054.911,158.554,-85.909,171.638,33.506,156.266
C06061=1054.905,158.297,-85.886,171.636,33.504,156.265
C06062=1054.899,158.038,-85.863,171.634,33.501,156.265
C06063=1054.892,157.781,-85.841,171.632,33.499,156.264
C06064=1054.887,157.532,-85.819,171.630,33.496,156.264
C06065=1054.880,157.283,-85.796,171.627,33.494,156.263
C06066=1054.874,157.034,-85.775,171.625,33.491,156.263
C06067=1054.869,156.785,-85.753,171.623,33.489,156.263
C06068=1054.863,156.537,-85.730,171.622,33.487,156.262
C06069=1054.857,156.288,-85.709,171.620,33.484,156.262
C06070=1054.851,156.039,-85.686,171.618,33.482,156.261
C06071=1054.845,155.789,-85.664,171.616,33.479,156.261
C06072=1054.839,155.540,-85.642,171.614,33.476,156.261
C06073=1054.834,155.292,-85.620,171.612,33.474,156.260
C06074=1054.827,155.043,-85.598,171.610,33.471,156.260
C06075=1054.821,154.794,-85.577,171.608,33.469,156.259
C06076=1054.815,154.545,-85.554,171.606,33.467,156.259
C06077=1054.809,154.296,-85.532,171.604,33.464,156.258
C06078=1054.804,154.047,-85.511,171.602,33.462,156.258
C06079=1054.798,153.798,-85.489,171.601,33.459,156.258
C06080=1054.791,153.549,-85.467,171.599,33.457,156.257
C06081=1054.786,153.300,-85.445,171.597,33.455,156.257
C06082=1054.780,153.051,-85.423,171.595,33.452,156.256
C06083=1054.774,152.802,-85.402,171.593,33.449,156.256
C06084=1054.767,152.525,-85.377,171.591,33.447,156.255
C06085=1054.761,152.249,-85.353,171.589,33.444,156.255
C06086=1054.754,151.973,-85.329,171.587,33.441,156.254
C06087=1054.748,151.697,-85.305,171.585,33.439,156.254
C06088=1054.741,151.448,-85.282,171.583,33.436,156.254
C06089=1054.735,151.199,-85.261,171.581,33.434,156.253
C06090=1054.730,150.950,-85.239,171.579,33.432,156.253
C06091=1054.724,150.701,-85.217,171.577,33.429,156.252
C06092=1054.718,150.452,-85.196,171.575,33.426,156.252
C06093=1054.712,150.203,-85.174,171.573,33.424,156.252
C06094=1054.706,149.955,-85.152,171.571,33.421,156.251
C06095=1054.700,149.706,-85.130,171.570,33.419,156.251
C06096=1054.693,149.456,-85.109,171.568,33.417,156.250
C06097=1054.689,149.208,-85.087,171.566,33.414,156.250
C06098=1054.682,148.958,-85.065,171.564,33.412,156.249
C06099=1054.676,148.709,-85.044,171.562,33.409,156.249
C06100=1054.670,148.460,-85.022,171.560,33.407,156.249
C06101=1054.664,148.211,-85.001,171.558,33.405,156.248
C06102=1054.658,147.962,-84.979,171.556,33.402,156.248
C06103=1054.652,147.713,-84.957,171.554,33.400,156.247
C06104=1054.647,147.464,-84.936,171.552,33.397,156.247
C06105=1054.640,147.215,-84.915,171.550,33.395,156.247
C06106=1054.634,146.966,-84.893,171.548,33.392,156.246
C06107=1054.628,146.717,-84.871,171.546,33.390,156.246
C06108=1054.623,146.468,-84.850,171.544,33.388,156.245
C06109=1054.616,146.219,-84.828,171.542,33.385,156.245
C06110=1054.610,145.970,-84.807,171.541,33.383,156.245
C06111=1054.605,145.721,-84.785,171.539,33.380,156.244
C06112=1054.599,145.472,-84.764,171.537,33.378,156.244
C06113=1054.592,145.223,-84.742,171.535,33.376,156.243
C06114=1054.587,144.975,-84.721,171.533,33.373,156.243
C06115=1054.581,144.725,-84.699,171.531,33.371,156.242
C06116=1054.574,144.476,-84.678,171.530,33.369,156.242
C06117=1054.569,144.227,-84.657,171.528,33.366,156.242
C06118=1054.562,143.978,-84.636,171.526,33.364,156.241
C06119=1054.556,143.729,-84.614,171.524,33.362,156.241
C06120=1054.551,143.480,-84.593,171.522,33.359,156.240
C06121=1054.544,143.231,-84.571,171.520,33.356,156.240
C06122=1054.538,142.982,-84.550,171.518,33.354,156.240
C06123=1054.533,142.733,-84.529,171.517,33.352,156.239
C06124=1054.526,142.448,-84.504,171.515,33.349,156.239
C06125=1054.519,142.163,-84.480,171.512,33.346,156.238
C06126=1054.513,141.878,-84.455,171.510,33.344,156.238
C06127=1054.506,141.593,-84.431,171.508,33.340,156.237
C06128=1054.499,141.343,-84.410,171.506,33.338,156.237
C06129=1054.494,141.095,-84.388,171.505,33.336,156.237
C06130=1054.488,140.846,-84.367,171.503,33.333,156.236
C06131=1054.482,140.597,-84.346,171.501,33.331,156.236
C06132=1054.476,140.347,-84.325,171.499,33.329,156.235
C06133=1054.469,140.098,-84.304,171.497,33.326,156.235
C06134=1054.464,139.850,-84.282,171.496,33.324,156.234
C06135=1054.458,139.600,-84.261,171.494,33.322,156.234
C06136=1054.452,139.352,-84.240,171.492,33.319,156.234
C06137=1054.446,139.102,-84.218,171.490,33.317,156.233
C06138=1054.440,138.853,-84.198,171.488,33.315,156.233
C06139=1054.434,138.604,-84.177,171.486,33.312,156.233
C06140=1054.428,138.355,-84.155,171.485,33.310,156.232
C06141=1054.423,138.106,-84.135,171.483,33.308,156.232
C06142=1054.416,137.857,-84.114,171.481,33.305,156.231
C06143=1054.410,137.609,-84.092,171.479,33.302,156.231
C06144=1054.404,137.359,-84.071,171.477,33.300,156.230
C06145=1054.399,137.110,-84.050,171.476,33.298,156.230
C06146=1054.392,136.861,-84.030,171.474,33.295,156.230
C06147=1054.386,136.612,-84.008,171.472,33.293,156.229
C06148=1054.380,136.363,-83.987,171.470,33.291,156.229
C06149=1054.374,136.114,-83.967,171.468,33.288,156.229
C06150=1054.368,135.865,-83.945,171.467,33.286,156.228
C06151=1054.362,135.615,-83.924,171.465,33.284,156.228
C06152=1054.356,135.367,-83.904,171.463,33.281,156.227
C06153=1054.350,135.117,-83.883,171.461,33.279,156.227
C06154=1054.345,134.869,-83.862,171.459,33.277,156.227
C06155=1054.338,134.620,-83.841,171.458,33.274,156.226
C06156=1054.332,134.371,-83.820,171.456,33.272,156.226
C06157=1054.326,134.121,-83.798,171.454,33.270,156.225
C06158=1054.320,133.873,-83.778,171.452,33.267,156.225
C06159=1054.314,133.623,-83.757,171.450,33.265,156.225
C06160=1054.309,133.374,-83.736,171.449,33.263,156.224
C06161=1054.302,133.125,-83.715,171.447,33.260,156.224
C06162=1054.297,132.876,-83.695,171.445,33.258,156.223
C06163=1054.290,132.627,-83.674,171.443,33.255,156.223
C06164=1054.285,132.378,-83.653,171.441,33.253,156.223
C06165=1054.279,132.128,-83.632,171.439,33.251,156.222
C06166=1054.272,131.880,-83.611,171.437,33.248,156.222
C06167=1054.267,131.630,-83.591,171.435,33.246,156.221
C06168=1054.260,131.382,-83.570,171.433,33.244,156.221
C06169=1054.254,131.132,-83.549,171.432,33.241,156.221
C06170=1054.248,130.884,-83.529,171.430,33.239,156.220
C06171=1054.242,130.634,-83.507,171.428,33.237,156.220
C06172=1054.236,130.386,-83.487,171.426,33.235,156.220
C06173=1054.230,130.136,-83.467,171.425,33.232,156.219
C06174=1054.224,129.888,-83.446,171.423,33.230,156.219
C06175=1054.218,129.638,-83.425,171.421,33.228,156.218
C06176=1054.212,129.389,-83.405,171.419,33.225,156.218
C06177=1054.205,129.140,-83.384,171.417,33.223,156.218
C06178=1054.199,128.891,-83.364,171.416,33.221,156.217
C06179=1054.193,128.642,-83.344,171.414,33.219,156.217
C06180=1054.188,128.393,-83.323,171.412,33.216,156.216
C06181=1054.181,128.144,-83.302,171.410,33.214,156.216
C06182=1054.175,127.895,-83.281,171.409,33.212,156.216
C06183=1054.169,127.646,-83.261,171.407,33.210,156.215
C06184=1054.162,127.397,-83.240,171.405,33.207,156.215
C06185=1054.157,127.148,-83.220,171.403,33.204,156.214
C06186=1054.151,126.898,-83.200,171.401,33.202,156.214
C06187=1054.145,126.649,-83.180,171.400,33.200,156.214
C06188=1054.138,126.364,-83.156,171.398,33.197,156.213
C06189=1054.131,126.079,-83.132,171.396,33.195,156.213
C06190=1054.124,125.793,-83.109,171.394,33.192,156.212
C06191=1054.117,125.509,-83.085,171.392,33.190,156.212
C06192=1054.111,125.259,-83.065,171.390,33.188,156.212
C06193=1054.105,125.010,-83.045,171.388,33.185,156.211
C06194=1054.099,124.760,-83.024,171.386,33.182,156.211
C06195=1054.093,124.512,-83.004,171.385,33.181,156.210
C06196=1054.087,124.263,-82.984,171.383,33.178,156.210
C06197=1054.081,124.014,-82.963,171.381,33.176,156.210
C06198=1054.075,123.765,-82.943,171.379,33.173,156.209
C06199=1054.069,123.516,-82.923,171.378,33.171,156.209
C06200=1054.063,123.266,-82.902,171.376,33.169,156.208
C06201=1054.057,123.017,-82.882,171.374,33.166,156.208
C06202=1054.050,122.768,-82.861,171.372,33.164,156.208
C06203=1054.045,122.519,-82.841,171.371,33.162,156.207
C06204=1054.039,122.270,-82.821,171.369,33.160,156.207
C06205=1054.032,122.020,-82.801,171.367,33.157,156.207
C06206=1054.027,121.771,-82.780,171.365,33.155,156.206
C06207=1054.021,121.522,-82.760,171.364,33.153,156.206
C06208=1054.014,121.274,-82.739,171.362,33.150,156.205
C06209=1054.008,121.025,-82.719,171.360,33.148,156.205
C06210=1054.003,120.776,-82.699,171.359,33.146,156.205
C06211=1053.997,120.527,-82.679,171.357,33.144,156.204
C06212=1053.990,120.277,-82.658,171.355,33.141,156.204
C06213=1053.985,120.028,-82.638,171.353,33.138,156.203
C06214=1053.979,119.779,-82.618,171.352,33.137,156.203
C06215=1053.972,119.530,-82.597,171.350,33.134,156.203
C06216=1053.966,119.281,-82.577,171.348,33.132,156.202
C06217=1053.961,119.032,-82.557,171.346,33.129,156.202
C06218=1053.956,118.782,-82.538,171.345,33.127,156.201
C06219=1053.949,118.533,-82.517,171.343,33.125,156.201
C06220=1053.943,118.284,-82.497,171.341,33.122,156.201
C06221=1053.938,118.035,-82.477,171.340,33.120,156.200
C06222=1053.932,117.786,-82.457,171.338,33.118,156.200
C06223=1053.925,117.537,-82.437,171.336,33.115,156.200
C06224=1053.920,117.288,-82.416,171.334,33.113,156.199
C06225=1053.914,117.039,-82.396,171.333,33.111,156.199
C06226=1053.908,116.790,-82.376,171.331,33.108,156.198
C06227=1053.901,116.540,-82.356,171.329,33.106,156.198
C06228=1053.896,116.291,-82.335,171.328,33.104,156.198
C06229=1053.890,116.042,-82.315,171.326,33.101,156.197
C06230=1053.884,115.793,-82.296,171.324,33.099,156.197
C06231=1053.878,115.544,-82.276,171.323,33.097,156.196
C06232=1053.872,115.294,-82.255,171.321,33.095,156.196
C06233=1053.867,115.046,-82.235,171.319,33.092,156.196
C06234=1053.861,114.797,-82.215,171.317,33.089,156.195
C06235=1053.855,114.548,-82.195,171.316,33.087,156.195
C06236=1053.849,114.299,-82.176,171.314,33.085,156.194
C06237=1053.843,114.049,-82.155,171.312,33.082,156.194
C06238=1053.837,113.800,-82.135,171.311,33.080,156.194
C06239=1053.831,113.551,-82.115,171.309,33.078,156.193
C06240=1053.825,113.302,-82.096,171.307,33.076,156.193
C06241=1053.819,113.052,-82.076,171.306,33.073,156.193
C06242=1053.813,112.803,-82.056,171.304,33.071,156.192
C06243=1053.807,112.554,-82.036,171.302,33.069,156.192
C06244=1053.801,112.305,-82.016,171.300,33.067,156.191
C06245=1053.795,112.056,-81.996,171.299,33.064,156.191
C06246=1053.788,111.807,-81.976,171.297,33.062,156.191
C06247=1053.783,111.557,-81.957,171.295,33.060,156.190
C06248=1053.777,111.308,-81.937,171.294,33.058,156.190
C06249=1053.771,111.060,-81.917,171.292,33.055,156.190
C06250=1053.765,110.810,-81.898,171.290,33.053,156.189
C06251=1053.758,110.561,-81.877,171.289,33.051,156.189
C06252=1053.752,110.276,-81.855,171.287,33.048,156.188
C06253=1053.744,109.990,-81.833,171.285,33.045,156.188
C06254=1053.738,109.705,-81.810,171.283,33.043,156.187
C06255=1053.730,109.420,-81.787,171.281,33.040,156.187
C06256=1053.725,109.170,-81.768,171.279,33.038,156.187
C06257=1053.719,108.921,-81.748,171.277,33.035,156.186
C06258=1053.713,108.673,-81.728,171.276,33.034,156.186
C06259=1053.706,108.423,-81.709,171.274,33.031,156.186
C06260=1053.700,108.174,-81.689,171.272,33.029,156.185
C06261=1053.694,107.924,-81.670,171.271,33.027,156.185
C06262=1053.688,107.676,-81.650,171.270,33.024,156.184
C06263=1053.682,107.426,-81.631,171.268,33.022,156.184
C06264=1053.676,107.177,-81.611,171.266,33.020,156.184
C06265=1053.669,106.928,-81.592,171.265,33.018,156.183
C06266=1053.663,106.679,-81.572,171.263,33.015,156.183
C06267=1053.658,106.429,-81.553,171.261,33.013,156.183
C06268=1053.652,106.181,-81.533,171.260,33.011,156.182
C06269=1053.646,105.931,-81.513,171.258,33.009,156.182
C06270=1053.640,105.682,-81.494,171.256,33.006,156.181
C06271=1053.633,105.433,-81.475,171.255,33.004,156.181
C06272=1053.627,105.184,-81.455,171.253,33.002,156.181
C06273=1053.621,104.934,-81.435,171.251,33.000,156.180
C06274=1053.615,104.685,-81.415,171.250,32.997,156.180
C06275=1053.610,104.436,-81.396,171.248,32.995,156.180
C06276=1053.603,104.188,-81.377,171.246,32.993,156.179
C06277=1053.597,103.938,-81.358,171.245,32.991,156.179
C06278=1053.591,103.689,-81.338,171.243,32.988,156.178
C06279=1053.585,103.440,-81.318,171.241,32.986,156.178
C06280=1053.580,103.190,-81.299,171.240,32.984,156.178
C06281=1053.573,102.942,-81.280,171.238,32.982,156.177
C06282=1053.567,102.692,-81.260,171.236,32.979,156.177
C06283=1053.562,102.443,-81.241,171.235,32.977,156.177
C06284=1053.556,102.194,-81.221,171.233,32.974,156.176
C06285=1053.550,101.945,-81.202,171.231,32.972,156.176
C06286=1053.544,101.696,-81.183,171.230,32.970,156.175
C06287=1053.538,101.447,-81.163,171.228,32.968,156.175
C06288=1053.531,101.197,-81.144,171.226,32.965,156.175
C06289=1053.526,100.947,-81.125,171.225,32.963,156.174
C06290=1053.520,100.698,-81.105,171.223,32.961,156.174
C06291=1053.513,100.449,-81.086,171.221,32.959,156.174
C06292=1053.507,100.200,-81.067,171.220,32.956,156.173
C06293=1053.501,99.951,-81.047,171.218,32.954,156.173
C06294=1053.495,99.702,-81.028,171.216,32.952,156.172
C06295=1053.489,99.453,-81.009,171.214,32.950,156.172
C06296=1053.483,99.203,-80.990,171.213,32.948,156.172
C06297=1053.476,98.955,-80.971,171.211,32.945,156.171
C06298=1053.470,98.705,-80.952,171.209,32.943,156.171
C06299=1053.465,98.456,-80.932,171.208,32.941,156.171
C06300=1053.458,98.207,-80.914,171.206,32.939,156.170
C06301=1053.453,97.957,-80.894,171.204,32.937,156.170
C06302=1053.446,97.709,-80.875,171.203,32.934,156.170
C06303=1053.440,97.460,-80.856,171.201,32.932,156.169
C06304=1053.434,97.210,-80.837,171.199,32.929,156.169
C06305=1053.428,96.961,-80.818,171.198,32.928,156.169
C06306=1053.422,96.712,-80.799,171.196,32.925,156.168
C06307=1053.416,96.462,-80.780,171.194,32.923,156.168
C06308=1053.409,96.214,-80.761,171.193,32.921,156.167
C06309=1053.404,95.965,-80.741,171.191,32.918,156.167
C06310=1053.397,95.715,-80.723,171.189,32.916,156.167
C06311=1053.391,95.466,-80.704,171.188,32.914,156.166
C06312=1053.386,95.217,-80.684,171.186,32.912,156.166
C06313=1053.379,94.967,-80.666,171.184,32.909,156.166
C06314=1053.374,94.718,-80.646,171.183,32.907,156.165
C06315=1053.367,94.469,-80.628,171.181,32.905,156.165
C06316=1053.360,94.183,-80.605,171.179,32.903,156.165
C06317=1053.353,93.898,-80.583,171.177,32.900,156.164
C06318=1053.346,93.613,-80.562,171.175,32.897,156.164
C06319=1053.340,93.328,-80.540,171.174,32.895,156.163
C06320=1053.333,93.078,-80.522,171.172,32.892,156.163
C06321=1053.327,92.829,-80.502,171.170,32.890,156.162
C06322=1053.321,92.580,-80.484,171.169,32.888,156.162
C06323=1053.315,92.330,-80.464,171.167,32.886,156.162
C06324=1053.309,92.081,-80.446,171.165,32.883,156.161
C06325=1053.303,91.832,-80.427,171.164,32.881,156.161
C06326=1053.297,91.583,-80.408,171.162,32.879,156.161
C06327=1053.291,91.333,-80.389,171.160,32.877,156.160
C06328=1053.285,91.084,-80.370,171.159,32.875,156.160
C06329=1053.280,90.835,-80.351,171.158,32.872,156.160
C06330=1053.273,90.586,-80.332,171.156,32.870,156.159
C06331=1053.268,90.337,-80.313,171.155,32.868,156.159
C06332=1053.261,90.088,-80.295,171.153,32.866,156.158
C06333=1053.255,89.839,-80.276,171.151,32.863,156.158
C06334=1053.248,89.590,-80.257,171.150,32.861,156.158
C06335=1053.243,89.339,-80.239,171.148,32.859,156.157
C06336=1053.236,89.090,-80.220,171.146,32.856,156.157
C06337=1053.230,88.841,-80.201,171.145,32.854,156.157
C06338=1053.224,88.592,-80.183,171.143,32.852,156.156
C06339=1053.218,88.343,-80.164,171.141,32.850,156.156
C06340=1053.211,88.094,-80.145,171.140,32.848,156.156
C06341=1053.205,87.844,-80.126,171.138,32.846,156.155
C06342=1053.199,87.595,-80.108,171.137,32.843,156.155
C06343=1053.194,87.346,-80.089,171.135,32.841,156.155
C06344=1053.187,87.097,-80.071,171.133,32.839,156.154
C06345=1053.181,86.848,-80.052,171.132,32.837,156.154
C06346=1053.175,86.599,-80.034,171.130,32.835,156.153
C06347=1053.169,86.349,-80.014,171.128,32.833,156.153
C06348=1053.163,86.099,-79.996,171.127,32.830,156.153
C06349=1053.156,85.850,-79.978,171.125,32.828,156.152
C06350=1053.150,85.601,-79.959,171.123,32.826,156.152
C06351=1053.144,85.353,-79.941,171.122,32.824,156.152
C06352=1053.138,85.103,-79.922,171.120,32.822,156.151
C06353=1053.132,84.854,-79.904,171.118,32.819,156.151
C06354=1053.126,84.604,-79.885,171.117,32.817,156.151
C06355=1053.119,84.355,-79.866,171.115,32.815,156.150
C06356=1053.114,84.106,-79.847,171.113,32.812,156.150
C06357=1053.108,83.856,-79.829,171.112,32.811,156.150
C06358=1053.102,83.608,-79.811,171.110,32.808,156.149
C06359=1053.095,83.359,-79.792,171.108,32.806,156.149
C06360=1053.089,83.109,-79.774,171.107,32.804,156.148
C06361=1053.084,82.859,-79.755,171.105,32.801,156.148
C06362=1053.077,82.610,-79.736,171.104,32.799,156.148
C06363=1053.072,82.361,-79.719,171.102,32.797,156.147
C06364=1053.065,82.112,-79.700,171.100,32.795,156.147
C06365=1053.059,81.863,-79.681,171.099,32.793,156.147
C06366=1053.053,81.613,-79.663,171.097,32.790,156.146
C06367=1053.047,81.364,-79.644,171.095,32.788,156.146
C06368=1053.041,81.115,-79.626,171.094,32.786,156.146
C06369=1053.035,80.866,-79.608,171.092,32.784,156.145
C06370=1053.029,80.617,-79.589,171.091,32.782,156.145
C06371=1053.022,80.367,-79.571,171.090,32.779,156.144
C06372=1053.017,80.118,-79.553,171.088,32.777,156.144
C06373=1053.011,79.869,-79.534,171.087,32.775,156.144
C06374=1053.005,79.619,-79.516,171.085,32.773,156.143
C06375=1052.998,79.370,-79.497,171.083,32.770,156.143
C06376=1052.993,79.122,-79.479,171.082,32.768,156.143
C06377=1052.986,78.872,-79.461,171.080,32.766,156.142
C06378=1052.981,78.623,-79.442,171.078,32.763,156.142
C06379=1052.975,78.373,-79.424,171.077,32.761,156.142
C06380=1052.967,78.088,-79.403,171.075,32.759,156.141
C06381=1052.960,77.802,-79.383,171.073,32.756,156.141
C06382=1052.954,77.517,-79.361,171.071,32.754,156.140
C06383=1052.946,77.231,-79.341,171.069,32.751,156.140
C06384=1052.940,76.982,-79.322,171.068,32.749,156.140
C06385=1052.934,76.733,-79.305,171.066,32.747,156.139
C06386=1052.928,76.484,-79.286,171.064,32.745,156.139
C06387=1052.922,76.234,-79.268,171.063,32.742,156.139
C06388=1052.916,75.985,-79.250,171.061,32.740,156.138
C06389=1052.910,75.736,-79.232,171.059,32.738,156.138
C06390=1052.904,75.486,-79.214,171.058,32.736,156.138
C06391=1052.897,75.237,-79.195,171.056,32.734,156.137
C06392=1052.891,74.987,-79.177,171.054,32.732,156.137
C06393=1052.885,74.739,-79.159,171.053,32.729,156.136
C06394=1052.879,74.490,-79.142,171.051,32.727,156.136
C06395=1052.872,74.240,-79.124,171.049,32.725,156.136
C06396=1052.867,73.991,-79.105,171.048,32.723,156.135
C06397=1052.860,73.742,-79.087,171.046,32.721,156.135
C06398=1052.854,73.493,-79.069,171.045,32.719,156.135
C06399=1052.848,73.243,-79.051,171.043,32.716,156.134
C06400=1052.842,72.994,-79.033,171.041,32.714,156.134
C06401=1052.836,72.745,-79.015,171.040,32.712,156.134
C06402=1052.830,72.495,-78.997,171.039,32.709,156.133
C06403=1052.824,72.246,-78.979,171.037,32.707,156.133
C06404=1052.818,71.997,-78.961,171.036,32.705,156.133
C06405=1052.811,71.747,-78.943,171.034,32.703,156.132
C06406=1052.806,71.498,-78.926,171.032,32.701,156.132
C06407=1052.799,71.249,-78.907,171.031,32.699,156.132
C06408=1052.793,70.999,-78.889,171.029,32.696,156.131
C06409=1052.787,70.750,-78.871,171.028,32.694,156.131
C06410=1052.781,70.501,-78.853,171.026,32.692,156.131
C06411=1052.775,70.252,-78.835,171.024,32.690,156.130
C06412=1052.769,70.003,-78.817,171.023,32.688,156.130
C06413=1052.763,69.753,-78.800,171.021,32.686,156.130
C06414=1052.756,69.504,-78.781,171.019,32.683,156.129
C06415=1052.751,69.255,-78.764,171.018,32.681,156.129
C06416=1052.744,69.005,-78.746,171.016,32.679,156.128
C06417=1052.738,68.756,-78.728,171.014,32.676,156.128
C06418=1052.732,68.507,-78.711,171.013,32.675,156.128
C06419=1052.726,68.258,-78.692,171.011,32.673,156.127
C06420=1052.720,68.009,-78.675,171.010,32.671,156.127
C06421=1052.713,67.759,-78.657,171.008,32.668,156.127
C06422=1052.707,67.509,-78.639,171.006,32.666,156.126
C06423=1052.702,67.260,-78.622,171.005,32.664,156.126
C06424=1052.696,67.011,-78.604,171.003,32.661,156.126
C06425=1052.688,66.762,-78.586,171.001,32.659,156.125
C06426=1052.683,66.513,-78.568,171.000,32.657,156.125
C06427=1052.677,66.263,-78.550,170.998,32.655,156.125
C06428=1052.670,66.014,-78.533,170.996,32.653,156.124
C06429=1052.664,65.765,-78.515,170.995,32.651,156.124
C06430=1052.658,65.515,-78.498,170.994,32.649,156.124
C06431=1052.653,65.266,-78.480,170.992,32.646,156.123
C06432=1052.646,65.016,-78.463,170.991,32.644,156.123
C06433=1052.640,64.768,-78.444,170.989,32.642,156.123
C06434=1052.634,64.518,-78.426,170.988,32.640,156.122
C06435=1052.627,64.269,-78.409,170.986,32.638,156.122
C06436=1052.622,64.020,-78.392,170.984,32.636,156.122
C06437=1052.615,63.770,-78.374,170.983,32.634,156.121
C06438=1052.609,63.521,-78.357,170.981,32.632,156.121
C06439=1052.602,63.272,-78.339,170.979,32.630,156.121
C06440=1052.596,63.022,-78.321,170.978,32.627,156.120
C06441=1052.590,62.773,-78.304,170.976,32.625,156.120
C06442=1052.584,62.524,-78.286,170.974,32.623,156.120
C06443=1052.577,62.274,-78.269,170.973,32.621,156.119
C06444=1052.571,61.989,-78.250,170.971,32.618,156.119
C06445=1052.563,61.703,-78.230,170.969,32.616,156.119
C06446=1052.556,61.418,-78.209,170.967,32.614,156.118
C06447=1052.549,61.132,-78.190,170.965,32.611,156.118
C06448=1052.542,60.883,-78.172,170.963,32.609,156.117
C06449=1052.536,60.634,-78.155,170.962,32.607,156.117
C06450=1052.529,60.384,-78.137,170.960,32.605,156.117
C06451=1052.524,60.135,-78.120,170.958,32.603,156.117
C06452=1052.517,59.885,-78.103,170.957,32.601,156.116
C06453=1052.510,59.636,-78.086,170.955,32.598,156.116
C06454=1052.505,59.387,-78.068,170.953,32.596,156.115
C06455=1052.498,59.137,-78.051,170.953,32.594,156.115
C06456=1052.493,58.888,-78.033,170.951,32.592,156.115
C06457=1052.486,58.639,-78.016,170.950,32.590,156.115
C06458=1052.479,58.390,-77.999,170.948,32.588,156.114
C06459=1052.474,58.140,-77.982,170.946,32.586,156.114
C06460=1052.467,57.891,-77.965,170.945,32.584,156.113
C06461=1052.461,57.641,-77.947,170.943,32.582,156.113
C06462=1052.455,57.392,-77.930,170.941,32.580,156.113
C06463=1052.448,57.143,-77.913,170.940,32.578,156.113
C06464=1052.443,56.894,-77.895,170.938,32.575,156.112
C06465=1052.436,56.644,-77.878,170.936,32.573,156.112
C06466=1052.431,56.395,-77.861,170.935,32.571,156.112
C06467=1052.424,56.145,-77.843,170.933,32.569,156.111
C06468=1052.417,55.897,-77.826,170.931,32.567,156.111
C06469=1052.411,55.647,-77.809,170.930,32.565,156.110
C06470=1052.405,55.398,-77.792,170.928,32.563,156.110
C06471=1052.399,55.148,-77.774,170.926,32.561,156.110
C06472=1052.393,54.899,-77.757,170.925,32.559,156.110
C06473=1052.386,54.650,-77.740,170.923,32.556,156.109
C06474=1052.381,54.400,-77.723,170.921,32.554,156.109
C06475=1052.374,54.151,-77.706,170.920,32.552,156.109
C06476=1052.368,53.902,-77.689,170.918,32.550,156.108
C06477=1052.362,53.652,-77.671,170.917,32.548,156.108
C06478=1052.356,53.403,-77.655,170.916,32.545,156.107
C06479=1052.350,53.153,-77.637,170.914,32.543,156.107
C06480=1052.343,52.904,-77.620,170.913,32.541,156.107
C06481=1052.337,52.655,-77.604,170.911,32.539,156.107
C06482=1052.331,52.405,-77.586,170.909,32.537,156.106
C06483=1052.325,52.157,-77.569,170.908,32.535,156.106
C06484=1052.318,51.906,-77.552,170.906,32.533,156.106
C06485=1052.313,51.657,-77.534,170.904,32.531,156.105
C06486=1052.307,51.409,-77.517,170.903,32.529,156.105
C06487=1052.300,51.159,-77.501,170.901,32.526,156.104
C06488=1052.295,50.910,-77.483,170.899,32.524,156.104
C06489=1052.288,50.660,-77.467,170.898,32.522,156.104
C06490=1052.282,50.411,-77.450,170.896,32.520,156.104
C06491=1052.276,50.162,-77.432,170.894,32.517,156.103
C06492=1052.270,49.912,-77.415,170.893,32.515,156.103
C06493=1052.263,49.663,-77.399,170.891,32.513,156.103
C06494=1052.258,49.414,-77.381,170.889,32.511,156.102
C06495=1052.251,49.164,-77.364,170.888,32.509,156.102
C06496=1052.245,48.915,-77.347,170.886,32.507,156.101
C06497=1052.239,48.665,-77.330,170.885,32.505,156.101
C06498=1052.233,48.416,-77.313,170.883,32.503,156.101
C06499=1052.227,48.167,-77.297,170.882,32.500,156.100
C06500=1052.221,47.917,-77.279,170.881,32.498,156.100
C06501=1052.215,47.668,-77.263,170.879,32.496,156.100
C06502=1052.209,47.419,-77.246,170.877,32.494,156.100
C06503=1052.203,47.169,-77.229,170.876,32.492,156.099
C06504=1052.197,46.920,-77.212,170.874,32.489,156.099
C06505=1052.191,46.671,-77.195,170.872,32.487,156.098
C06506=1052.185,46.421,-77.178,170.871,32.485,156.098
C06507=1052.179,46.171,-77.161,170.869,32.483,156.098
C06508=1052.172,45.885,-77.141,170.867,32.481,156.097
C06509=1052.165,45.601,-77.122,170.865,32.478,156.097
C06510=1052.158,45.314,-77.103,170.863,32.475,156.097
C06511=1052.151,45.028,-77.083,170.862,32.474,156.096
C06512=1052.145,44.779,-77.067,170.860,32.471,156.096
C06513=1052.139,44.530,-77.050,170.858,32.469,156.096
C06514=1052.132,44.280,-77.033,170.857,32.467,156.095
C06515=1052.127,44.030,-77.016,170.855,32.464,156.095
C06516=1052.121,43.782,-76.999,170.853,32.462,156.095
C06517=1052.115,43.532,-76.983,170.852,32.460,156.094
C06518=1052.108,43.283,-76.966,170.851,32.458,156.094
C06519=1052.102,43.033,-76.949,170.849,32.456,156.094
C06520=1052.097,42.784,-76.933,170.848,32.454,156.093
C06521=1052.090,42.534,-76.915,170.846,32.452,156.093
C06522=1052.084,42.285,-76.899,170.844,32.449,156.093
C06523=1052.078,42.036,-76.883,170.843,32.448,156.092
C06524=1052.072,41.787,-76.866,170.841,32.445,156.092
C06525=1052.065,41.537,-76.849,170.839,32.443,156.092
C06526=1052.059,41.288,-76.833,170.838,32.442,156.091
C06527=1052.053,41.039,-76.816,170.836,32.439,156.091
C06528=1052.047,40.789,-76.799,170.834,32.437,156.091
C06529=1052.041,40.539,-76.783,170.833,32.435,156.090
C06530=1052.035,40.290,-76.767,170.831,32.433,156.090
C06531=1052.028,40.041,-76.750,170.829,32.431,156.090
C06532=1052.022,39.791,-76.733,170.828,32.429,156.089
C06533=1052.016,39.542,-76.717,170.826,32.427,156.089
C06534=1052.010,39.293,-76.700,170.824,32.424,156.089
C06535=1052.004,39.044,-76.684,170.823,32.422,156.088
C06536=1051.997,38.794,-76.667,170.821,32.420,156.088
C06537=1051.991,38.544,-76.651,170.820,32.418,156.088
C06538=1051.985,38.295,-76.635,170.819,32.416,156.087
C06539=1051.980,38.046,-76.617,170.817,32.414,156.087
C06540=1051.974,37.797,-76.601,170.815,32.411,156.087
C06541=1051.966,37.547,-76.585,170.814,32.409,156.086
C06542=1051.960,37.298,-76.568,170.812,32.407,156.086
C06543=1051.955,37.048,-76.552,170.810,32.405,156.086
C06544=1051.949,36.799,-76.536,170.809,32.403,156.086
C06545=1051.942,36.550,-76.519,170.807,32.401,156.085
C06546=1051.936,36.300,-76.502,170.805,32.399,156.085
C06547=1051.930,36.051,-76.486,170.804,32.397,156.085
C06548=1051.923,35.802,-76.470,170.802,32.395,156.084
C06549=1051.917,35.552,-76.454,170.800,32.393,156.084
C06550=1051.911,35.302,-76.438,170.798,32.391,156.084
C06551=1051.905,35.053,-76.421,170.797,32.389,156.083
C06552=1051.899,34.804,-76.405,170.795,32.387,156.083
C06553=1051.893,34.554,-76.389,170.793,32.385,156.083
C06554=1051.885,34.305,-76.372,170.792,32.383,156.082
C06555=1051.879,34.056,-76.356,170.791,32.381,156.082
C06556=1051.873,33.807,-76.340,170.789,32.379,156.082
C06557=1051.867,33.557,-76.323,170.788,32.376,156.081
C06558=1051.861,33.308,-76.307,170.786,32.374,156.081
C06559=1051.854,33.058,-76.291,170.784,32.372,156.081
C06560=1051.848,32.809,-76.275,170.783,32.370,156.081
C06561=1051.842,32.559,-76.258,170.781,32.368,156.080
C06562=1051.836,32.310,-76.242,170.779,32.366,156.080
C06563=1051.830,32.061,-76.226,170.778,32.364,156.080
C06564=1051.824,31.811,-76.210,170.776,32.362,156.079
C06565=1051.817,31.562,-76.194,170.774,32.360,156.079
C06566=1051.811,31.312,-76.177,170.773,32.358,156.079
C06567=1051.805,31.063,-76.161,170.771,32.356,156.078
C06568=1051.799,30.814,-76.145,170.769,32.354,156.078
C06569=1051.793,30.564,-76.129,170.767,32.352,156.078
C06570=1051.787,30.315,-76.113,170.766,32.350,156.078
C06571=1051.781,30.066,-76.097,170.764,32.348,156.077
C06572=1051.773,29.780,-76.078,170.763,32.345,156.077
C06573=1051.766,29.494,-76.060,170.761,32.343,156.077
C06574=1051.759,29.207,-76.042,170.759,32.341,156.076
C06575=1051.753,28.922,-76.024,170.757,32.338,156.076
C06576=1051.747,28.672,-76.007,170.756,32.336,156.075
C06577=1051.740,28.422,-75.991,170.754,32.334,156.075
C06578=1051.733,28.173,-75.975,170.752,32.332,156.075
C06579=1051.727,27.924,-75.959,170.751,32.330,156.074
C06580=1051.721,27.675,-75.943,170.749,32.328,156.074
C06581=1051.715,27.425,-75.927,170.747,32.326,156.074
C06582=1051.709,27.176,-75.911,170.745,32.324,156.074
C06583=1051.703,26.926,-75.895,170.744,32.322,156.073
C06584=1051.696,26.677,-75.879,170.742,32.320,156.073
C06585=1051.690,26.428,-75.863,170.740,32.318,156.073
C06586=1051.683,26.178,-75.847,170.739,32.316,156.072
C06587=1051.678,25.928,-75.832,170.737,32.314,156.072
C06588=1051.672,25.679,-75.815,170.736,32.312,156.072
C06589=1051.665,25.430,-75.800,170.734,32.310,156.072
C06590=1051.659,25.180,-75.783,170.733,32.308,156.071
C06591=1051.652,24.931,-75.768,170.731,32.306,156.071
C06592=1051.647,24.681,-75.752,170.729,32.304,156.071
C06593=1051.640,24.432,-75.737,170.728,32.302,156.070
C06594=1051.634,24.183,-75.720,170.726,32.300,156.070
C06595=1051.628,23.934,-75.704,170.724,32.298,156.070
C06596=1051.622,23.684,-75.689,170.723,32.296,156.069
C06597=1051.616,23.435,-75.673,170.721,32.294,156.069
C06598=1051.609,23.186,-75.657,170.719,32.292,156.069
C06599=1051.603,22.936,-75.642,170.717,32.290,156.069
C06600=1051.597,22.687,-75.626,170.716,32.288,156.068
C06601=1051.591,22.437,-75.610,170.714,32.286,156.068
C06602=1051.585,22.187,-75.594,170.712,32.284,156.068
C06603=1051.578,21.938,-75.579,170.711,32.282,156.067
C06604=1051.572,21.688,-75.562,170.710,32.280,156.067
C06605=1051.565,21.438,-75.547,170.708,32.278,156.067
C06606=1051.560,21.189,-75.531,170.706,32.276,156.066
C06607=1051.553,20.940,-75.515,170.705,32.274,156.066
C06608=1051.547,20.690,-75.500,170.703,32.272,156.066
C06609=1051.540,20.441,-75.484,170.701,32.270,156.066
C06610=1051.535,20.192,-75.468,170.700,32.268,156.065
C06611=1051.528,19.942,-75.453,170.698,32.266,156.065
C06612=1051.522,19.693,-75.436,170.696,32.264,156.065
C06613=1051.516,19.443,-75.421,170.694,32.261,156.064
C06614=1051.510,19.194,-75.405,170.693,32.260,156.064
C06615=1051.503,18.944,-75.390,170.691,32.258,156.064
C06616=1051.497,18.695,-75.375,170.689,32.256,156.064
C06617=1051.491,18.446,-75.358,170.687,32.254,156.063
C06618=1051.484,18.196,-75.343,170.686,32.252,156.063
C06619=1051.479,17.947,-75.328,170.684,32.250,156.063
C06620=1051.473,17.698,-75.313,170.683,32.248,156.062
C06621=1051.466,17.449,-75.297,170.681,32.246,156.062
C06622=1051.460,17.199,-75.281,170.680,32.244,156.062
C06623=1051.454,16.950,-75.266,170.678,32.242,156.061
C06624=1051.448,16.700,-75.250,170.676,32.240,156.061
C06625=1051.441,16.451,-75.234,170.675,32.238,156.061
C06626=1051.435,16.201,-75.220,170.673,32.236,156.061
C06627=1051.429,15.952,-75.203,170.671,32.234,156.060
C06628=1051.423,15.702,-75.188,170.669,32.232,156.060
C06629=1051.417,15.452,-75.173,170.668,32.230,156.060
C06630=1051.410,15.203,-75.157,170.666,32.228,156.059
C06631=1051.404,14.953,-75.142,170.664,32.226,156.059
C06632=1051.398,14.704,-75.126,170.662,32.224,156.059
C06633=1051.392,14.454,-75.111,170.661,32.222,156.059
C06634=1051.386,14.205,-75.095,170.659,32.220,156.058
C06635=1051.379,13.955,-75.080,170.658,32.218,156.058
C06636=1051.372,13.671,-75.062,170.656,32.216,156.058
C06637=1051.365,13.387,-75.046,170.654,32.214,156.057
C06638=1051.357,13.101,-75.028,170.652,32.212,156.057
C06639=1051.350,12.817,-75.011,170.650,32.210,156.057
C06640=1051.343,12.568,-74.995,170.648,32.207,156.056
C06641=1051.338,12.318,-74.980,170.647,32.206,156.056
C06642=1051.331,12.068,-74.965,170.645,32.204,156.056
C06643=1051.325,11.819,-74.949,170.643,32.202,156.056
C06644=1051.318,11.570,-74.934,170.641,32.200,156.055
C06645=1051.313,11.321,-74.919,170.640,32.198,156.055
C06646=1051.306,11.072,-74.904,170.638,32.196,156.055
C06647=1051.300,10.822,-74.889,170.636,32.194,156.055
C06648=1051.294,10.572,-74.873,170.634,32.192,156.054
C06649=1051.288,10.322,-74.858,170.634,32.190,156.054
C06650=1051.281,10.073,-74.843,170.632,32.189,156.054
C06651=1051.274,9.824,-74.828,170.630,32.187,156.054
C06652=1051.268,9.574,-74.813,170.628,32.185,156.053
C06653=1051.262,9.324,-74.798,170.626,32.183,156.053
C06654=1051.256,9.076,-74.783,170.625,32.181,156.053
C06655=1051.250,8.826,-74.767,170.623,32.179,156.052
C06656=1051.244,8.576,-74.752,170.621,32.177,156.052
C06657=1051.237,8.327,-74.737,170.619,32.175,156.052
C06658=1051.231,8.077,-74.722,170.618,32.173,156.052
C06659=1051.224,7.828,-74.706,170.616,32.172,156.051
C06660=1051.218,7.578,-74.692,170.614,32.170,156.051
C06661=1051.212,7.329,-74.677,170.612,32.168,156.051
C06662=1051.206,7.080,-74.662,170.611,32.166,156.050
C06663=1051.199,6.830,-74.647,170.610,32.164,156.050
C06664=1051.194,6.580,-74.632,170.608,32.162,156.050
C06665=1051.187,6.331,-74.616,170.606,32.160,156.050
C06666=1051.180,6.081,-74.601,170.604,32.158,156.049
C06667=1051.175,5.832,-74.586,170.603,32.157,156.049
C06668=1051.168,5.583,-74.571,170.601,32.154,156.049
C06669=1051.162,5.333,-74.556,170.599,32.152,156.049
C06670=1051.156,5.083,-74.542,170.597,32.150,156.048
C06671=1051.149,4.834,-74.527,170.596,32.148,156.048
C06672=1051.143,4.585,-74.512,170.594,32.147,156.048
C06673=1051.137,4.335,-74.497,170.592,32.145,156.048
C06674=1051.131,4.086,-74.482,170.590,32.143,156.047
C06675=1051.125,3.836,-74.466,170.588,32.141,156.047
C06676=1051.119,3.587,-74.451,170.587,32.139,156.047
C06677=1051.112,3.338,-74.436,170.586,32.137,156.046
C06678=1051.106,3.088,-74.421,170.584,32.135,156.046
C06679=1051.100,2.838,-74.406,170.582,32.133,156.046
C06680=1051.094,2.589,-74.392,170.580,32.132,156.046
C06681=1051.088,2.340,-74.377,170.579,32.130,156.045
C06682=1051.081,2.090,-74.362,170.577,32.128,156.045
C06683=1051.075,1.840,-74.347,170.575,32.125,156.045
C06684=1051.069,1.591,-74.332,170.573,32.124,156.045
C06685=1051.063,1.342,-74.317,170.572,32.122,156.044
C06686=1051.056,1.092,-74.303,170.570,32.120,156.044
C06687=1051.050,0.843,-74.288,170.568,32.118,156.044
C06688=1051.044,0.593,-74.273,170.566,32.116,156.044
C06689=1051.038,0.344,-74.258,170.564,32.114,156.043
C06690=1051.032,0.094,-74.243,170.563,32.112,156.043
C06691=1051.026,-0.155,-74.228,170.562,32.110,156.043
C06692=1051.020,-0.405,-74.213,170.560,32.108,156.042
C06693=1051.014,-0.655,-74.199,170.558,32.107,156.042
C06694=1051.008,-0.904,-74.184,170.556,32.105,156.042
C06695=1051.002,-1.154,-74.169,170.555,32.103,156.042
C06696=1050.995,-1.403,-74.154,170.553,32.101,156.041
C06697=1050.989,-1.652,-74.140,170.551,32.099,156.041
C06698=1050.983,-1.902,-74.125,170.549,32.097,156.041
C06699=1050.977,-2.152,-74.110,170.547,32.095,156.041
C06700=1050.970,-2.434,-74.093,170.545,32.093,156.040
C06701=1050.963,-2.717,-74.077,170.543,32.091,156.040
C06702=1050.956,-2.999,-74.060,170.541,32.089,156.040
C06703=1050.949,-3.281,-74.043,170.540,32.087,156.039
C06704=1050.943,-3.532,-74.029,170.539,32.085,156.039
C06705=1050.937,-3.781,-74.014,170.537,32.083,156.039
C06706=1050.930,-4.031,-73.999,170.535,32.081,156.039
C06707=1050.924,-4.280,-73.985,170.533,32.079,156.038
C06708=1050.918,-4.530,-73.971,170.531,32.078,156.038
C06709=1050.911,-4.780,-73.956,170.529,32.075,156.038
C06710=1050.906,-5.029,-73.941,170.528,32.074,156.038
C06711=1050.899,-5.278,-73.927,170.526,32.072,156.037
C06712=1050.892,-5.528,-73.913,170.524,32.071,156.037
C06713=1050.887,-5.777,-73.898,170.522,32.068,156.037
C06714=1050.880,-6.027,-73.884,170.520,32.066,156.037
C06715=1050.873,-6.276,-73.869,170.518,32.065,156.036
C06716=1050.868,-6.526,-73.855,170.517,32.063,156.036
C06717=1050.861,-6.775,-73.840,170.516,32.061,156.036
C06718=1050.854,-7.025,-73.826,170.514,32.059,156.036
C06719=1050.849,-7.274,-73.812,170.512,32.058,156.035
C06720=1050.842,-7.524,-73.797,170.510,32.056,156.035
C06721=1050.837,-7.773,-73.782,170.508,32.054,156.035
C06722=1050.830,-8.023,-73.769,170.507,32.052,156.035
C06723=1050.823,-8.273,-73.754,170.505,32.050,156.034
C06724=1050.818,-8.522,-73.739,170.503,32.049,156.034
C06725=1050.811,-8.772,-73.726,170.501,32.047,156.034
C06726=1050.805,-9.020,-73.711,170.499,32.045,156.034
C06727=1050.799,-9.270,-73.696,170.497,32.043,156.033
C06728=1050.793,-9.520,-73.682,170.495,32.042,156.033
C06729=1050.786,-9.769,-73.668,170.494,32.040,156.033
C06730=1050.780,-10.019,-73.654,170.493,32.038,156.033
C06731=1050.774,-10.268,-73.639,170.491,32.036,156.032
C06732=1050.767,-10.518,-73.625,170.489,32.034,156.032
C06733=1050.762,-10.767,-73.611,170.487,32.033,156.032
C06734=1050.755,-11.017,-73.596,170.485,32.030,156.032
C06735=1050.748,-11.267,-73.582,170.484,32.029,156.032
C06736=1050.743,-11.516,-73.568,170.482,32.027,156.031
C06737=1050.736,-11.766,-73.554,170.480,32.026,156.031
C06738=1050.730,-12.015,-73.540,170.478,32.023,156.031
C06739=1050.724,-12.264,-73.525,170.476,32.022,156.031
C06740=1050.718,-12.514,-73.511,170.474,32.020,156.030
C06741=1050.711,-12.763,-73.496,170.472,32.018,156.030
C06742=1050.705,-13.013,-73.483,170.471,32.016,156.030
C06743=1050.699,-13.262,-73.468,170.470,32.014,156.030
C06744=1050.693,-13.512,-73.454,170.468,32.013,156.029
C06745=1050.687,-13.761,-73.439,170.466,32.011,156.029
C06746=1050.681,-14.011,-73.425,170.464,32.009,156.029
C06747=1050.674,-14.261,-73.412,170.462,32.007,156.029
C06748=1050.668,-14.510,-73.397,170.460,32.006,156.028
C06749=1050.662,-14.760,-73.383,170.459,32.004,156.028
C06750=1050.656,-15.009,-73.369,170.457,32.002,156.028
C06751=1050.650,-15.259,-73.355,170.455,32.000,156.028
C06752=1050.643,-15.508,-73.341,170.453,31.999,156.027
C06753=1050.637,-15.758,-73.327,170.451,31.997,156.027
C06754=1050.631,-16.007,-73.313,170.449,31.995,156.027
C06755=1050.625,-16.257,-73.298,170.448,31.994,156.027
C06756=1050.618,-16.506,-73.285,170.446,31.992,156.027
C06757=1050.612,-16.757,-73.271,170.445,31.990,156.026
C06758=1050.606,-17.005,-73.257,170.443,31.989,156.026
C06759=1050.600,-17.255,-73.243,170.441,31.987,156.026
C06760=1050.593,-17.504,-73.229,170.439,31.985,156.026
C06761=1050.586,-17.754,-73.215,170.437,31.983,156.025
C06762=1050.581,-18.004,-73.201,170.435,31.982,156.025
C06763=1050.574,-18.254,-73.188,170.433,31.980,156.025
C06764=1050.567,-18.535,-73.172,170.431,31.978,156.025
C06765=1050.560,-18.816,-73.156,170.429,31.976,156.025
C06766=1050.553,-19.097,-73.140,170.427,31.974,156.024
C06767=1050.546,-19.378,-73.125,170.425,31.972,156.024
C06768=1050.539,-19.627,-73.110,170.424,31.971,156.024
C06769=1050.533,-19.877,-73.097,170.422,31.969,156.024
C06770=1050.528,-20.126,-73.083,170.420,31.967,156.023
C06771=1050.521,-20.376,-73.069,170.418,31.965,156.023
C06772=1050.515,-20.625,-73.055,170.416,31.964,156.023
C06773=1050.508,-20.875,-73.041,170.414,31.962,156.023
C06774=1050.503,-21.125,-73.027,170.413,31.960,156.022
C06775=1050.496,-21.375,-73.014,170.411,31.959,156.022
C06776=1050.489,-21.623,-73.000,170.409,31.957,156.022
C06777=1050.484,-21.873,-72.986,170.407,31.955,156.022
C06778=1050.477,-22.123,-72.972,170.405,31.954,156.022
C06779=1050.471,-22.372,-72.959,170.403,31.952,156.021
C06780=1050.465,-22.622,-72.945,170.402,31.950,156.021
C06781=1050.459,-22.872,-72.932,170.400,31.949,156.021
C06782=1050.453,-23.121,-72.917,170.398,31.947,156.021
C06783=1050.446,-23.371,-72.903,170.396,31.945,156.021
C06784=1050.440,-23.620,-72.890,170.395,31.944,156.020
C06785=1050.434,-23.869,-72.876,170.393,31.942,156.020
C06786=1050.427,-24.119,-72.863,170.391,31.940,156.020
C06787=1050.422,-24.369,-72.849,170.389,31.939,156.020
C06788=1050.416,-24.618,-72.835,170.387,31.937,156.019
C06789=1050.409,-24.868,-72.821,170.385,31.935,156.019
C06790=1050.403,-25.117,-72.807,170.383,31.934,156.019
C06791=1050.397,-25.366,-72.794,170.381,31.931,156.019
C06792=1050.390,-25.616,-72.780,170.380,31.930,156.019
C06793=1050.385,-25.866,-72.766,170.378,31.929,156.018
C06794=1050.378,-26.115,-72.753,170.376,31.926,156.018
C06795=1050.372,-26.365,-72.740,170.374,31.925,156.018
C06796=1050.366,-26.615,-72.726,170.373,31.924,156.018
C06797=1050.360,-26.864,-72.712,170.371,31.922,156.018
C06798=1050.353,-27.114,-72.699,170.369,31.920,156.017
C06799=1050.347,-27.363,-72.685,170.367,31.918,156.017
C06800=1050.341,-27.613,-72.672,170.365,31.917,156.017
C06801=1050.335,-27.863,-72.658,170.363,31.916,156.017
C06802=1050.328,-28.112,-72.645,170.361,31.914,156.017
C06803=1050.322,-28.361,-72.631,170.359,31.912,156.016
C06804=1050.315,-28.611,-72.618,170.357,31.910,156.016
C06805=1050.309,-28.860,-72.605,170.356,31.909,156.016
C06806=1050.303,-29.110,-72.591,170.354,31.907,156.016
C06807=1050.297,-29.360,-72.577,170.352,31.906,156.016
C06808=1050.291,-29.609,-72.564,170.350,31.905,156.015
C06809=1050.284,-29.859,-72.550,170.348,31.902,156.015
C06810=1050.278,-30.109,-72.537,170.346,31.901,156.015
C06811=1050.272,-30.358,-72.524,170.344,31.899,156.015
C06812=1050.265,-30.608,-72.511,170.343,31.898,156.015
C06813=1050.259,-30.857,-72.498,170.341,31.897,156.014
C06814=1050.252,-31.107,-72.484,170.339,31.895,156.014
C06815=1050.246,-31.356,-72.471,170.337,31.893,156.014
C06816=1050.241,-31.606,-72.457,170.335,31.892,156.014
C06817=1050.234,-31.856,-72.443,170.334,31.890,156.014
C06818=1050.228,-32.105,-72.430,170.332,31.889,156.013
C06819=1050.222,-32.355,-72.418,170.330,31.887,156.013
C06820=1050.216,-32.604,-72.404,170.328,31.886,156.013
C06821=1050.209,-32.854,-72.391,170.326,31.884,156.013
C06822=1050.203,-33.103,-72.377,170.324,31.882,156.013
C06823=1050.196,-33.353,-72.364,170.322,31.880,156.013
C06824=1050.190,-33.602,-72.352,170.320,31.879,156.012
C06825=1050.184,-33.852,-72.338,170.318,31.877,156.012
C06826=1050.177,-34.102,-72.325,170.316,31.876,156.012
C06827=1050.172,-34.351,-72.311,170.314,31.875,156.012
C06828=1050.165,-34.631,-72.296,170.312,31.872,156.012
C06829=1050.158,-34.911,-72.281,170.311,31.871,156.011
C06830=1050.151,-35.192,-72.267,170.309,31.869,156.011
C06831=1050.144,-35.472,-72.252,170.306,31.867,156.011
C06832=1050.137,-35.722,-72.239,170.304,31.866,156.011
C06833=1050.131,-35.971,-72.225,170.302,31.864,156.011
C06834=1050.125,-36.221,-72.213,170.301,31.863,156.010
C06835=1050.120,-36.471,-72.199,170.299,31.861,156.010
C06836=1050.113,-36.720,-72.186,170.297,31.860,156.010
C06837=1050.107,-36.969,-72.173,170.295,31.858,156.010
C06838=1050.101,-37.220,-72.160,170.293,31.856,156.010
C06839=1050.094,-37.469,-72.146,170.291,31.855,156.009
C06840=1050.088,-37.719,-72.133,170.289,31.853,156.009
C06841=1050.082,-37.968,-72.120,170.288,31.852,156.009
C06842=1050.076,-38.218,-72.107,170.286,31.850,156.009
C06843=1050.070,-38.467,-72.094,170.284,31.849,156.009
C06844=1050.064,-38.717,-72.081,170.282,31.847,156.009
C06845=1050.057,-38.967,-72.068,170.280,31.846,156.008
C06846=1050.051,-39.217,-72.055,170.278,31.844,156.008
C06847=1050.044,-39.466,-72.043,170.276,31.843,156.008
C06848=1050.038,-39.715,-72.029,170.274,31.841,156.008
C06849=1050.032,-39.965,-72.017,170.272,31.840,156.008
C06850=1050.026,-40.214,-72.003,170.270,31.838,156.008
C06851=1050.019,-40.465,-71.991,170.268,31.837,156.007
C06852=1050.013,-40.714,-71.977,170.266,31.835,156.007
C06853=1050.007,-40.964,-71.965,170.265,31.834,156.007
C06854=1050.000,-41.213,-71.952,170.263,31.832,156.007
C06855=1049.994,-41.463,-71.939,170.261,31.831,156.007
C06856=1049.988,-41.712,-71.926,170.259,31.830,156.007
C06857=1049.982,-41.962,-71.914,170.257,31.829,156.006
C06858=1049.975,-42.211,-71.901,170.255,31.827,156.006
C06859=1049.969,-42.461,-71.888,170.253,31.826,156.006
C06860=1049.963,-42.711,-71.875,170.251,31.824,156.006
C06861=1049.957,-42.960,-71.862,170.249,31.823,156.006
C06862=1049.951,-43.210,-71.849,170.247,31.821,156.006
C06863=1049.945,-43.460,-71.836,170.245,31.820,156.005
C06864=1049.938,-43.709,-71.824,170.243,31.818,156.005
C06865=1049.932,-43.958,-71.811,170.242,31.817,156.005
C06866=1049.926,-44.208,-71.798,170.240,31.815,156.005
C06867=1049.920,-44.458,-71.785,170.238,31.814,156.005
C06868=1049.913,-44.707,-71.773,170.236,31.813,156.005
C06869=1049.907,-44.956,-71.760,170.234,31.811,156.004
C06870=1049.901,-45.206,-71.748,170.232,31.810,156.004
C06871=1049.895,-45.456,-71.734,170.230,31.808,156.004
C06872=1049.889,-45.705,-71.722,170.228,31.807,156.004
C06873=1049.882,-45.955,-71.710,170.226,31.805,156.004
C06874=1049.876,-46.204,-71.697,170.224,31.804,156.004
C06875=1049.870,-46.454,-71.684,170.222,31.802,156.003
C06876=1049.864,-46.703,-71.671,170.220,31.801,156.003
C06877=1049.857,-46.953,-71.659,170.219,31.800,156.003
C06878=1049.851,-47.203,-71.646,170.217,31.798,156.003
C06879=1049.845,-47.452,-71.633,170.215,31.797,156.003
C06880=1049.839,-47.702,-71.620,170.213,31.795,156.003
C06881=1049.833,-47.952,-71.608,170.211,31.794,156.003
C06882=1049.826,-48.201,-71.595,170.209,31.792,156.002
C06883=1049.820,-48.451,-71.583,170.206,31.791,156.002
C06884=1049.814,-48.701,-71.570,170.204,31.790,156.002
C06885=1049.808,-48.951,-71.557,170.202,31.788,156.002
C06886=1049.802,-49.199,-71.545,170.200,31.787,156.002
C06887=1049.796,-49.449,-71.532,170.198,31.785,156.002
C06888=1049.790,-49.699,-71.520,170.196,31.784,156.002
C06889=1049.784,-49.949,-71.507,170.195,31.782,156.001
C06890=1049.777,-50.198,-71.494,170.193,31.782,156.001
C06891=1049.771,-50.448,-71.482,170.191,31.780,156.001
C06892=1049.764,-50.729,-71.468,170.189,31.779,156.001
C06893=1049.756,-51.010,-71.454,170.187,31.777,156.001
C06894=1049.749,-51.291,-71.440,170.184,31.775,156.001
C06895=1049.742,-51.571,-71.426,170.182,31.774,156.000
C06896=1049.736,-51.821,-71.414,170.180,31.773,156.000
C06897=1049.729,-52.070,-71.402,170.178,31.772,156.000
C06898=1049.723,-52.320,-71.389,170.176,31.771,156.000
C06899=1049.717,-52.570,-71.377,170.174,31.769,156.000
C06900=1049.711,-52.820,-71.365,170.172,31.768,156.000
C06901=1049.704,-53.069,-71.353,170.171,31.767,156.000
C06902=1049.697,-53.318,-71.340,170.169,31.765,156.000
C06903=1049.691,-53.568,-71.328,170.166,31.764,156.000
C06904=1049.685,-53.818,-71.316,170.164,31.763,155.999
C06905=1049.679,-54.068,-71.303,170.162,31.761,155.999
C06906=1049.672,-54.317,-71.291,170.160,31.760,155.999
C06907=1049.665,-54.567,-71.279,170.158,31.759,155.999
C06908=1049.660,-54.817,-71.267,170.156,31.758,155.999
C06909=1049.653,-55.066,-71.255,170.154,31.757,155.999
C06910=1049.647,-55.316,-71.242,170.152,31.755,155.999
C06911=1049.640,-55.566,-71.230,170.150,31.754,155.999
C06912=1049.634,-55.814,-71.219,170.148,31.753,155.998
C06913=1049.628,-56.064,-71.206,170.146,31.752,155.998
C06914=1049.622,-56.314,-71.194,170.145,31.750,155.998
C06915=1049.616,-56.564,-71.182,170.143,31.749,155.998
C06916=1049.609,-56.813,-71.170,170.141,31.748,155.998
C06917=1049.603,-57.063,-71.158,170.138,31.746,155.998
C06918=1049.597,-57.313,-71.145,170.136,31.745,155.998
C06919=1049.590,-57.562,-71.133,170.134,31.744,155.998
C06920=1049.583,-57.812,-71.121,170.132,31.743,155.997
C06921=1049.577,-58.062,-71.109,170.130,31.741,155.997
C06922=1049.571,-58.311,-71.097,170.128,31.741,155.997
C06923=1049.565,-58.561,-71.084,170.126,31.739,155.997
C06924=1049.559,-58.810,-71.073,170.124,31.738,155.997
C06925=1049.552,-59.060,-71.061,170.122,31.737,155.997
C06926=1049.546,-59.310,-71.048,170.121,31.736,155.997
C06927=1049.540,-59.559,-71.036,170.119,31.734,155.997
C06928=1049.534,-59.809,-71.025,170.117,31.733,155.997
C06929=1049.528,-60.059,-71.013,170.114,31.732,155.996
C06930=1049.521,-60.308,-71.001,170.112,31.731,155.996
C06931=1049.515,-60.558,-70.989,170.110,31.729,155.996
C06932=1049.509,-60.808,-70.976,170.108,31.729,155.996
C06933=1049.502,-61.057,-70.964,170.106,31.727,155.996
C06934=1049.496,-61.306,-70.953,170.104,31.726,155.996
C06935=1049.490,-61.556,-70.940,170.102,31.725,155.996
C06936=1049.484,-61.806,-70.929,170.100,31.724,155.996
C06937=1049.477,-62.056,-70.917,170.098,31.722,155.996
C06938=1049.472,-62.305,-70.905,170.096,31.721,155.995
C06939=1049.465,-62.554,-70.893,170.095,31.720,155.995
C06940=1049.459,-62.804,-70.881,170.092,31.719,155.995
C06941=1049.453,-63.055,-70.869,170.090,31.717,155.995
C06942=1049.446,-63.304,-70.857,170.088,31.716,155.995
C06943=1049.440,-63.553,-70.845,170.086,31.715,155.995
C06944=1049.434,-63.803,-70.833,170.084,31.714,155.995
C06945=1049.428,-64.053,-70.822,170.082,31.713,155.995
C06946=1049.421,-64.303,-70.810,170.080,31.712,155.995
C06947=1049.416,-64.552,-70.797,170.078,31.710,155.994
C06948=1049.409,-64.801,-70.785,170.076,31.709,155.994
C06949=1049.403,-65.052,-70.774,170.074,31.708,155.994
C06950=1049.397,-65.300,-70.763,170.071,31.707,155.994
C06951=1049.391,-65.550,-70.750,170.070,31.706,155.994
C06952=1049.385,-65.800,-70.738,170.068,31.704,155.994
C06953=1049.378,-66.050,-70.727,170.066,31.704,155.994
C06954=1049.373,-66.299,-70.715,170.064,31.702,155.994
C06955=1049.366,-66.549,-70.703,170.062,31.701,155.994
C06956=1049.359,-66.832,-70.690,170.060,31.700,155.994
C06957=1049.352,-67.114,-70.676,170.057,31.699,155.993
C06958=1049.346,-67.395,-70.663,170.055,31.697,155.993
C06959=1049.339,-67.677,-70.650,170.052,31.695,155.993
C06960=1049.333,-67.927,-70.638,170.050,31.695,155.993
C06961=1049.327,-68.177,-70.627,170.048,31.694,155.993
C06962=1049.320,-68.426,-70.615,170.046,31.692,155.993
C06963=1049.314,-68.676,-70.603,170.045,31.691,155.993
C06964=1049.309,-68.926,-70.591,170.043,31.690,155.993
C06965=1049.302,-69.175,-70.579,170.041,31.689,155.993
C06966=1049.296,-69.425,-70.568,170.039,31.688,155.993
C06967=1049.290,-69.674,-70.557,170.036,31.686,155.992
C06968=1049.284,-69.924,-70.544,170.034,31.686,155.992
C06969=1049.277,-70.174,-70.533,170.032,31.685,155.992
C06970=1049.271,-70.423,-70.521,170.030,31.683,155.992
C06971=1049.265,-70.673,-70.510,170.028,31.682,155.992
C06972=1049.260,-70.923,-70.498,170.026,31.681,155.992
C06973=1049.253,-71.173,-70.487,170.024,31.680,155.992
C06974=1049.247,-71.422,-70.475,170.022,31.679,155.992
C06975=1049.241,-71.672,-70.464,170.021,31.677,155.992
C06976=1049.235,-71.922,-70.451,170.018,31.676,155.992
C06977=1049.229,-72.171,-70.440,170.016,31.676,155.992
C06978=1049.223,-72.421,-70.428,170.014,31.674,155.991
C06979=1049.217,-72.670,-70.417,170.012,31.673,155.991
C06980=1049.211,-72.920,-70.405,170.010,31.672,155.991
C06981=1049.205,-73.170,-70.394,170.008,31.671,155.991
C06982=1049.199,-73.419,-70.382,170.006,31.670,155.991
C06983=1049.192,-73.669,-70.371,170.004,31.669,155.991
C06984=1049.187,-73.919,-70.359,170.001,31.667,155.991
C06985=1049.181,-74.169,-70.347,169.999,31.666,155.991
C06986=1049.175,-74.418,-70.337,169.997,31.666,155.991
C06987=1049.168,-74.668,-70.325,169.995,31.665,155.991
C06988=1049.162,-74.917,-70.314,169.994,31.664,155.991
C06989=1049.155,-75.167,-70.303,169.992,31.663,155.991
C06990=1049.149,-75.417,-70.291,169.990,31.662,155.991
C06991=1049.143,-75.666,-70.280,169.987,31.660,155.990
C06992=1049.136,-75.916,-70.268,169.985,31.659,155.990
C06993=1049.131,-76.165,-70.257,169.983,31.659,155.990
C06994=1049.124,-76.415,-70.246,169.981,31.658,155.990
C06995=1049.118,-76.664,-70.235,169.979,31.657,155.990
C06996=1049.112,-76.915,-70.223,169.977,31.656,155.990
C06997=1049.106,-77.164,-70.212,169.974,31.655,155.990
C06998=1049.100,-77.414,-70.201,169.972,31.654,155.990
C06999=1049.094,-77.663,-70.190,169.970,31.653,155.990
C07000=1049.087,-77.913,-70.178,169.968,31.652,155.990
C07001=1049.081,-78.163,-70.167,169.967,31.651,155.990
C07002=1049.075,-78.412,-70.155,169.965,31.650,155.990
C07003=1049.069,-78.663,-70.144,169.962,31.649,155.990
C07004=1049.063,-78.912,-70.133,169.960,31.648,155.990
C07005=1049.057,-79.162,-70.122,169.958,31.647,155.990
C07006=1049.051,-79.411,-70.111,169.956,31.646,155.989
C07007=1049.045,-79.661,-70.100,169.954,31.645,155.989
C07008=1049.038,-79.911,-70.088,169.952,31.644,155.989
C07009=1049.031,-80.161,-70.078,169.949,31.643,155.989
C07010=1049.026,-80.410,-70.067,169.947,31.642,155.989
C07011=1049.019,-80.660,-70.056,169.945,31.642,155.989
C07012=1049.013,-80.909,-70.044,169.943,31.641,155.989
C07013=1049.006,-81.159,-70.033,169.941,31.640,155.989
C07014=1049.000,-81.409,-70.023,169.940,31.639,155.989
C07015=1048.994,-81.659,-70.011,169.937,31.638,155.989
C07016=1048.988,-81.908,-70.000,169.935,31.637,155.989
C07017=1048.981,-82.158,-69.990,169.933,31.637,155.989
C07018=1048.976,-82.408,-69.979,169.931,31.636,155.989
C07019=1048.969,-82.657,-69.967,169.929,31.635,155.989
C07020=1048.962,-82.942,-69.955,169.926,31.634,155.989
C07021=1048.954,-83.226,-69.943,169.924,31.633,155.989
C07022=1048.947,-83.510,-69.930,169.921,31.632,155.989
C07023=1048.941,-83.794,-69.918,169.919,31.631,155.989
C07024=1048.934,-84.044,-69.907,169.916,31.630,155.989
C07025=1048.928,-84.293,-69.896,169.914,31.629,155.989
C07026=1048.921,-84.543,-69.885,169.912,31.628,155.989
C07027=1048.915,-84.793,-69.874,169.911,31.627,155.989
C07028=1048.910,-85.042,-69.863,169.909,31.627,155.989
C07029=1048.903,-85.292,-69.852,169.906,31.626,155.989
C07030=1048.897,-85.541,-69.842,169.904,31.625,155.989
C07031=1048.891,-85.792,-69.830,169.902,31.624,155.988
C07032=1048.885,-86.041,-69.819,169.900,31.623,155.988
C07033=1048.878,-86.290,-69.809,169.898,31.623,155.988
C07034=1048.872,-86.541,-69.798,169.896,31.622,155.988
C07035=1048.866,-86.790,-69.787,169.893,31.621,155.988
C07036=1048.859,-87.041,-69.777,169.891,31.620,155.988
C07037=1048.854,-87.290,-69.766,169.889,31.620,155.988
C07038=1048.848,-87.540,-69.755,169.887,31.619,155.988
C07039=1048.841,-87.789,-69.745,169.885,31.618,155.988
C07040=1048.835,-88.039,-69.734,169.882,31.617,155.988
C07041=1048.829,-88.288,-69.723,169.881,31.616,155.988
C07042=1048.822,-88.538,-69.712,169.879,31.616,155.988
C07043=1048.817,-88.788,-69.701,169.877,31.615,155.988
C07044=1048.810,-89.038,-69.690,169.875,31.614,155.988
C07045=1048.804,-89.287,-69.680,169.872,31.613,155.988
C07046=1048.798,-89.537,-69.669,169.870,31.612,155.988
C07047=1048.791,-89.786,-69.658,169.868,31.612,155.988
C07048=1048.786,-90.037,-69.648,169.866,31.611,155.988
C07049=1048.780,-90.286,-69.637,169.863,31.610,155.988
C07050=1048.773,-90.535,-69.627,169.861,31.609,155.988
C07051=1048.767,-90.785,-69.616,169.859,31.609,155.988
C07052=1048.761,-91.035,-69.605,169.857,31.608,155.988
C07053=1048.755,-91.284,-69.595,169.855,31.607,155.988
C07054=1048.749,-91.535,-69.584,169.852,31.606,155.988
C07055=1048.743,-91.784,-69.573,169.851,31.605,155.988
C07056=1048.737,-92.034,-69.563,169.849,31.605,155.988
C07057=1048.730,-92.284,-69.552,169.847,31.604,155.988
C07058=1048.724,-92.533,-69.541,169.845,31.603,155.988
C07059=1048.718,-92.783,-69.531,169.842,31.602,155.988
C07060=1048.713,-93.033,-69.520,169.840,31.602,155.988
C07061=1048.705,-93.282,-69.510,169.838,31.601,155.988
C07062=1048.700,-93.532,-69.499,169.836,31.600,155.988
C07063=1048.694,-93.782,-69.489,169.834,31.600,155.988
C07064=1048.688,-94.031,-69.478,169.831,31.599,155.988
C07065=1048.682,-94.281,-69.468,169.829,31.598,155.988
C07066=1048.675,-94.531,-69.457,169.827,31.598,155.988
C07067=1048.670,-94.781,-69.447,169.825,31.597,155.988
C07068=1048.663,-95.030,-69.436,169.823,31.596,155.988
C07069=1048.657,-95.279,-69.426,169.820,31.596,155.988
C07070=1048.651,-95.530,-69.415,169.819,31.595,155.988
C07071=1048.645,-95.779,-69.405,169.817,31.594,155.988
C07072=1048.639,-96.029,-69.394,169.815,31.594,155.988
C07073=1048.633,-96.279,-69.384,169.812,31.593,155.988
C07074=1048.627,-96.528,-69.373,169.810,31.592,155.988
C07075=1048.621,-96.778,-69.362,169.808,31.591,155.988
C07076=1048.615,-97.028,-69.353,169.806,31.591,155.988
C07077=1048.609,-97.278,-69.342,169.804,31.590,155.988
C07078=1048.603,-97.527,-69.332,169.801,31.589,155.988
C07079=1048.597,-97.777,-69.321,169.799,31.588,155.988
C07080=1048.590,-98.027,-69.311,169.797,31.588,155.988
C07081=1048.584,-98.277,-69.301,169.795,31.588,155.988
C07082=1048.578,-98.526,-69.290,169.792,31.587,155.988
C07083=1048.572,-98.776,-69.281,169.790,31.587,155.988
C07084=1048.564,-99.063,-69.269,169.788,31.586,155.988
C07085=1048.557,-99.349,-69.257,169.786,31.585,155.988
C07086=1048.550,-99.636,-69.245,169.783,31.584,155.988
C07087=1048.544,-99.922,-69.234,169.781,31.584,155.988
C07088=1048.537,-100.171,-69.223,169.779,31.583,155.988
C07089=1048.532,-100.421,-69.213,169.776,31.583,155.988
C07090=1048.525,-100.671,-69.203,169.774,31.582,155.988
C07091=1048.518,-100.921,-69.193,169.772,31.581,155.988
C07092=1048.513,-101.171,-69.182,169.770,31.581,155.988
C07093=1048.507,-101.420,-69.173,169.767,31.580,155.988
C07094=1048.500,-101.670,-69.162,169.765,31.580,155.988
C07095=1048.495,-101.920,-69.152,169.763,31.579,155.988
C07096=1048.488,-102.170,-69.142,169.761,31.579,155.988
C07097=1048.481,-102.419,-69.132,169.758,31.578,155.988
C07098=1048.476,-102.669,-69.121,169.756,31.577,155.988
C07099=1048.469,-102.919,-69.111,169.754,31.577,155.988
C07100=1048.463,-103.168,-69.102,169.753,31.576,155.988
C07101=1048.457,-103.418,-69.092,169.750,31.576,155.988
C07102=1048.451,-103.668,-69.081,169.748,31.576,155.988
C07103=1048.445,-103.917,-69.071,169.746,31.575,155.988
C07104=1048.439,-104.167,-69.062,169.744,31.574,155.988
C07105=1048.433,-104.417,-69.051,169.741,31.574,155.988
C07106=1048.426,-104.667,-69.041,169.739,31.573,155.988
C07107=1048.420,-104.917,-69.031,169.737,31.573,155.988
C07108=1048.414,-105.166,-69.022,169.735,31.573,155.988
C07109=1048.408,-105.416,-69.011,169.732,31.572,155.988
C07110=1048.402,-105.666,-69.001,169.730,31.571,155.988
C07111=1048.396,-105.915,-68.992,169.728,31.571,155.988
C07112=1048.389,-106.165,-68.981,169.726,31.571,155.988
C07113=1048.384,-106.415,-68.971,169.723,31.570,155.988
C07114=1048.378,-106.664,-68.962,169.721,31.570,155.988
C07115=1048.372,-106.914,-68.952,169.719,31.569,155.988
C07116=1048.365,-107.163,-68.942,169.718,31.568,155.988
C07117=1048.360,-107.414,-68.932,169.715,31.568,155.989
C07118=1048.353,-107.663,-68.922,169.713,31.568,155.989
C07119=1048.347,-107.913,-68.913,169.711,31.567,155.989
C07120=1048.341,-108.162,-68.902,169.709,31.567,155.989
C07121=1048.335,-108.412,-68.893,169.706,31.566,155.989
C07122=1048.328,-108.662,-68.883,169.704,31.566,155.989
C07123=1048.322,-108.912,-68.874,169.702,31.566,155.989
C07124=1048.316,-109.161,-68.863,169.699,31.565,155.989
C07125=1048.310,-109.411,-68.853,169.697,31.565,155.989
C07126=1048.304,-109.661,-68.844,169.695,31.565,155.989
C07127=1048.298,-109.911,-68.834,169.693,31.564,155.989
C07128=1048.292,-110.160,-68.824,169.690,31.563,155.989
C07129=1048.286,-110.410,-68.815,169.688,31.563,155.989
C07130=1048.279,-110.659,-68.805,169.686,31.563,155.989
C07131=1048.273,-110.909,-68.795,169.684,31.563,155.989
C07132=1048.267,-111.159,-68.785,169.682,31.562,155.989
C07133=1048.261,-111.409,-68.776,169.680,31.562,155.989
C07134=1048.255,-111.659,-68.766,169.678,31.562,155.989
C07135=1048.249,-111.909,-68.756,169.675,31.561,155.989
C07136=1048.243,-112.159,-68.747,169.673,31.561,155.990
C07137=1048.237,-112.408,-68.737,169.671,31.560,155.989
C07138=1048.231,-112.658,-68.727,169.669,31.560,155.990
C07139=1048.224,-112.907,-68.717,169.666,31.559,155.990
C07140=1048.218,-113.157,-68.708,169.664,31.559,155.990
C07141=1048.212,-113.407,-68.698,169.662,31.559,155.990
C07142=1048.206,-113.657,-68.688,169.660,31.559,155.990
C07143=1048.199,-113.906,-68.679,169.657,31.558,155.990
C07144=1048.193,-114.156,-68.669,169.655,31.558,155.990
C07145=1048.187,-114.406,-68.660,169.653,31.558,155.990
C07146=1048.181,-114.656,-68.650,169.650,31.557,155.990
C07147=1048.175,-114.906,-68.641,169.648,31.557,155.990
C07148=1048.169,-115.134,-68.632,169.646,31.557,155.990
C07149=1048.164,-115.362,-68.624,169.644,31.556,155.990
C07150=1048.158,-115.590,-68.615,169.643,31.556,155.990
C07151=1048.153,-115.819,-68.605,169.641,31.556,155.990
C07152=1048.147,-116.047,-68.597,169.639,31.556,155.990
C07153=1048.142,-116.275,-68.588,169.637,31.555,155.990
C07154=1048.136,-116.504,-68.580,169.635,31.555,155.991
C07155=1048.130,-116.732,-68.571,169.632,31.555,155.991
C07156=1048.124,-116.982,-68.562,169.630,31.554,155.991
C07157=1048.118,-117.232,-68.552,169.628,31.554,155.991
C07158=1048.112,-117.482,-68.543,169.626,31.554,155.991
C07159=1048.106,-117.731,-68.533,169.623,31.554,155.991
C07160=1048.100,-117.980,-68.524,169.621,31.554,155.991
C07161=1048.094,-118.230,-68.514,169.619,31.554,155.991
C07162=1048.087,-118.480,-68.505,169.616,31.553,155.991
C07163=1048.081,-118.730,-68.497,169.614,31.553,155.991
C07164=1048.073,-119.058,-68.484,169.611,31.552,155.991
C07165=1048.065,-119.386,-68.472,169.608,31.553,155.992
C07166=1048.057,-119.715,-68.460,169.605,31.552,155.992
C07167=1048.049,-120.043,-68.448,169.602,31.552,155.992
C07168=1048.043,-120.293,-68.438,169.601,31.552,155.992
C07169=1048.037,-120.543,-68.428,169.598,31.551,155.992
C07170=1048.031,-120.792,-68.419,169.596,31.551,155.992
C07171=1048.025,-121.042,-68.410,169.594,31.551,155.992
C07172=1048.019,-121.292,-68.401,169.592,31.551,155.992
C07173=1048.013,-121.542,-68.391,169.589,31.551,155.992
C07174=1048.006,-121.792,-68.382,169.587,31.550,155.992
C07175=1048.000,-122.041,-68.373,169.585,31.550,155.992
C07176=1047.994,-122.291,-68.363,169.582,31.550,155.993
C07177=1047.988,-122.541,-68.355,169.580,31.550,155.993
C07178=1047.982,-122.791,-68.345,169.578,31.550,155.993
C07179=1047.976,-123.041,-68.335,169.575,31.549,155.993
C07180=1047.970,-123.289,-68.327,169.573,31.550,155.993
C07181=1047.964,-123.540,-68.318,169.571,31.549,155.993
C07182=1047.958,-123.790,-68.308,169.569,31.549,155.993
C07183=1047.951,-124.039,-68.299,169.566,31.549,155.993
C07184=1047.946,-124.289,-68.290,169.564,31.549,155.993
C07185=1047.939,-124.539,-68.281,169.562,31.549,155.993
C07186=1047.933,-124.788,-68.272,169.559,31.549,155.993
C07187=1047.927,-125.039,-68.263,169.557,31.549,155.994
C07188=1047.921,-125.289,-68.253,169.555,31.549,155.994
C07189=1047.915,-125.537,-68.245,169.553,31.548,155.994
C07190=1047.909,-125.788,-68.236,169.551,31.549,155.994
C07191=1047.903,-126.038,-68.226,169.549,31.548,155.994
C07192=1047.896,-126.287,-68.217,169.547,31.548,155.994
C07193=1047.890,-126.537,-68.209,169.544,31.548,155.994
C07194=1047.884,-126.787,-68.199,169.542,31.548,155.994
C07195=1047.878,-127.037,-68.191,169.540,31.548,155.994
C07196=1047.872,-127.286,-68.182,169.537,31.548,155.995
C07197=1047.866,-127.536,-68.172,169.535,31.548,155.995
C07198=1047.859,-127.786,-68.164,169.533,31.548,155.995
C07199=1047.855,-128.035,-68.154,169.530,31.548,155.995
C07200=1047.850,-128.285,-68.144,169.528,31.547,155.995
C07201=1047.846,-128.534,-68.134,169.526,31.545,155.995
C07202=1047.844,-128.785,-68.122,169.524,31.544,155.994
C07203=1047.842,-129.035,-68.110,169.523,31.541,155.994
C07204=1047.842,-129.285,-68.098,169.522,31.538,155.994
C07205=1047.843,-129.536,-68.084,169.520,31.535,155.993
C07206=1047.844,-129.786,-68.071,169.519,31.532,155.993
C07207=1047.847,-130.035,-68.057,169.517,31.528,155.992
C07208=1047.850,-130.287,-68.041,169.516,31.522,155.991
C07209=1047.855,-130.537,-68.025,169.516,31.518,155.990
C07210=1047.860,-130.788,-68.009,169.515,31.512,155.990
C07211=1047.867,-131.038,-67.992,169.514,31.506,155.989
C07212=1047.507,-131.061,-68.225,169.468,31.680,156.021
C07213=1047.500,-130.811,-68.243,169.469,31.686,156.022
C07214=1047.495,-130.561,-68.259,169.470,31.692,156.023
C07215=1047.490,-130.310,-68.274,169.470,31.697,156.024
C07216=1047.487,-130.060,-68.289,169.471,31.701,156.024
C07217=1047.484,-129.810,-68.305,169.473,31.705,156.025
C07218=1047.482,-129.559,-68.318,169.474,31.709,156.025
C07219=1047.482,-129.309,-68.331,169.476,31.712,156.026
C07220=1047.482,-129.058,-68.344,169.478,31.715,156.026
C07221=1047.483,-128.808,-68.356,169.478,31.717,156.027
C07222=1047.486,-128.558,-68.367,169.480,31.719,156.027
C07223=1047.489,-128.308,-68.378,169.482,31.721,156.027
C07224=1047.494,-128.059,-68.388,169.484,31.721,156.027
C07225=1047.499,-127.809,-68.398,169.487,31.722,156.027
C07226=1047.505,-127.559,-68.407,169.489,31.722,156.027
C07227=1047.511,-127.310,-68.415,169.491,31.722,156.027
C07228=1047.517,-127.060,-68.425,169.494,31.722,156.027
C07229=1047.523,-126.810,-68.434,169.496,31.722,156.026
C07230=1047.529,-126.561,-68.442,169.498,31.722,156.026
C07231=1047.536,-126.311,-68.452,169.501,31.722,156.026
C07232=1047.541,-126.061,-68.461,169.503,31.722,156.026
C07233=1047.548,-125.811,-68.470,169.505,31.722,156.026
C07234=1047.554,-125.562,-68.478,169.508,31.722,156.026
C07235=1047.560,-125.312,-68.488,169.510,31.722,156.026
C07236=1047.567,-125.062,-68.497,169.512,31.722,156.026
C07237=1047.573,-124.812,-68.506,169.514,31.722,156.026
C07238=1047.578,-124.563,-68.515,169.517,31.723,156.026
C07239=1047.584,-124.313,-68.524,169.518,31.723,156.025
C07240=1047.591,-124.063,-68.533,169.520,31.722,156.025
C07241=1047.597,-123.813,-68.542,169.523,31.723,156.025
C07242=1047.603,-123.564,-68.551,169.525,31.723,156.025
